// TIA Portal project "Project20" (V19)

(* hardware
DEVICE "S7-1200 station_1"  S7-1200 Station
   slot 0: "Rack_0"  S7-1200 Rack  Rack  V1.0
   slot 1: "PLC_1"  CPU 1215C DC/DC/DC  6ES7 215-1AG40-0XB0  V4.5
*)

// ===== PLC "PLC_1"  CPU 1215C DC/DC/DC =====

VAR_GLOBAL   // PLC tag table "Default tag table"
   "Contactor_Bomba1" AT %Q0.0 : Bool;
   "Contactor_Bomba2" AT %Q0.1 : Bool;
   "Contactor_Bomba3" AT %Q0.2 : Bool;
   "Contactor_Bomba4" AT %Q0.3 : Bool;
   "Contactor_Inyectora" AT %Q0.4 : Bool;
   "Contactor_Bandeja" AT %Q0.5 : Bool;
   "System_Byte" AT %MB1 : Byte;
   "FirstScan" AT %M1.0 : Bool;
   "DiagStatusUpdate" AT %M1.1 : Bool;
   "AlwaysTRUE" AT %M1.2 : Bool;
   "AlwaysFALSE" AT %M1.3 : Bool;
   "Clock_Byte" AT %MB8000 : Byte;
   "Clock_10Hz" AT %M8000.0 : Bool;
   "Clock_5Hz" AT %M8000.1 : Bool;
   "Clock_2.5Hz" AT %M8000.2 : Bool;
   "Clock_2Hz" AT %M8000.3 : Bool;
   "Clock_1.25Hz" AT %M8000.4 : Bool;
   "Clock_1Hz" AT %M8000.5 : Bool;
   "Clock_0.625Hz" AT %M8000.6 : Bool;
   "Clock_0.5Hz" AT %M8000.7 : Bool;
   "Valvula_Entrada_TanqueEntrada" AT %M0.0 : Bool;
   "Valvula_Entrada_TanqueSec1" AT %M0.1 : Bool;
   "Valvula_Entrada_TanqueSec2" AT %M0.2 : Bool;
   "Valvula_Salida_TanqueEntrada" AT %M0.3 : Bool;
   "Valvula_Salida_TanqueSec1" AT %M0.4 : Bool;
   "Valvula_Salida_TanqueSec2" AT %M0.5 : Bool;
   "Pulsador_Bomba1" AT %M0.6 : Bool;
   "Pulsador_Bomba2" AT %M0.7 : Bool;
   "Pulsador_Bomba3" AT %M2.0 : Bool;
   "Pulsador_Bomba4" AT %M2.1 : Bool;
   "Marca_Interruptor" AT %M2.2 : Bool;
   "Marca_Seccionador" AT %M2.3 : Bool;
   "Apertura_Interruptor" AT %M2.4 : Bool;
   "Apertura_Seccionador" AT %M2.5 : Bool;
   "Comando_Llenadora" AT %M2.6 : Bool;
   "Comando_Empacadora" AT %M2.7 : Bool;
END_VAR

TYPE "Datos_Jugos"
VERSION : 0.1
   STRUCT
      Agua : Real;
      Jarabe : Real;
      Manzana : Real;
      Banana : Real;
      Pera : Real;
   END_STRUCT;
END_TYPE

TYPE "Motor_Bomba"
VERSION : 0.1
   STRUCT
      Tension : Array[0..3] of Real;
      Corriente : Real;
      Velocidad : Real;
   END_STRUCT;
END_TYPE

DATA_BLOCK "DB_Llenadora3Botellas"   // DB1
{ S7_Optimized_Access := 'TRUE' }
VERSION : 0.1
// stored: InstanceOfName FB_Llenadora3Botellas
"FB_Llenadora3Botellas"
BEGIN
END_DATA_BLOCK

DATA_BLOCK "DB_Insumos"   // DB8
{ S7_Optimized_Access := 'TRUE' }
VERSION : 0.1
   VAR
      ContajeDinInsumos : Int;
      NivelBotella1 : Int := 0;
      NivelBotella2 : Int := 0;
      NivelBotella3 : Int := 0;
      RecetaActual : Int;
      Jugos : "Datos_Jugos";
   END_VAR
BEGIN
END_DATA_BLOCK

DATA_BLOCK "DB_Fallas"   // DB9
{ S7_Optimized_Access := 'TRUE' }
VERSION : 0.1
BEGIN
END_DATA_BLOCK

DATA_BLOCK "DB_MotorBomba1"   // DB10
{ S7_Optimized_Access := 'TRUE' }
VERSION : 0.1
// stored: InstanceOfName FB_MotorBomba
"FB_MotorBomba"
BEGIN
END_DATA_BLOCK

DATA_BLOCK "DB_MotorBomba2"   // DB11
{ S7_Optimized_Access := 'TRUE' }
VERSION : 0.1
// stored: InstanceOfName FB_MotorBomba
"FB_MotorBomba"
BEGIN
END_DATA_BLOCK

DATA_BLOCK "DB_TanqueEntrada"   // DB12
{ S7_Optimized_Access := 'TRUE' }
VERSION : 0.1
// stored: InstanceOfName FB_Tanque
"FB_Tanque"
BEGIN
END_DATA_BLOCK

DATA_BLOCK "DB_TanqueSec1"   // DB13
{ S7_Optimized_Access := 'TRUE' }
VERSION : 0.1
// stored: InstanceOfName FB_Tanque
"FB_Tanque"
BEGIN
END_DATA_BLOCK

DATA_BLOCK "DB_TanqueSec2"   // DB14
{ S7_Optimized_Access := 'TRUE' }
VERSION : 0.1
// stored: InstanceOfName FB_Tanque
"FB_Tanque"
BEGIN
END_DATA_BLOCK

DATA_BLOCK "DB_MotorBomba3"   // DB15
{ S7_Optimized_Access := 'TRUE' }
VERSION : 0.1
// stored: InstanceOfName FB_MotorBomba
"FB_MotorBomba"
BEGIN
END_DATA_BLOCK

DATA_BLOCK "DB_MotorBomba4"   // DB18
{ S7_Optimized_Access := 'TRUE' }
VERSION : 0.1
// stored: InstanceOfName FB_MotorBomba
"FB_MotorBomba"
BEGIN
END_DATA_BLOCK

DATA_BLOCK "DB_LecturaTensiones"   // DB20
{ S7_Optimized_Access := 'FALSE' }
VERSION : 0.1
   VAR
      Off : Bool;
      Modo : USInt;
      Data_Addr : UDInt := 43020;
      Data_Length : UDInt := 10;
      Connect : TCON_IP_v4;
      Buffer : Array[0..9] of Real;
      TensionSalida : Array[0..2] of Real;
      TensionEscalada : Array[0..5] of Real;
      Accionar_Interruptor : Bool;
      Accionar_Seccionador : Bool;
      Cierre_Interruptor : Bool;
      Cierre_Seccionador : Bool;
      Estado_Interruptor : Bool;
      Estado_Seccionador : Bool;
      ArrayVacio : Array[0..9] of Real;
   END_VAR
BEGIN
   Connect.RemoteAddress.ADDR[1] := 192;
   Connect.RemoteAddress.ADDR[2] := 168;
   Connect.RemoteAddress.ADDR[3] := 13;
   Connect.RemoteAddress.ADDR[4] := 68;
   Connect.InterfaceId := 64;
   Connect.ID := 1;
   Connect.ConnectionType := 11;
   Connect.ActiveEstablished := TRUE;
   Connect.RemotePort := 502;
END_DATA_BLOCK

DATA_BLOCK "DB_LecturaMotores"   // DB21
{ S7_Optimized_Access := 'TRUE' }
VERSION : 0.1
   VAR
      MotorBomba1 : "Motor_Bomba";
      MotorBomba2 : "Motor_Bomba";
      MotorBomba3 : "Motor_Bomba";
      MotorBomba4 : "Motor_Bomba";
      Angulo : Int;
      TensionSalida : Array[0..2] of Real;
   END_VAR
BEGIN
END_DATA_BLOCK

DATA_BLOCK "DB_LecturaMedidor"   // DB38
{ S7_Optimized_Access := 'FALSE' }
VERSION : 0.1
// stored: InstanceOfName FB_LecturaMedidor
"FB_LecturaMedidor"
BEGIN
END_DATA_BLOCK

DATA_BLOCK "DB_LecturaCorrientes"   // DB39
{ S7_Optimized_Access := 'FALSE' }
VERSION : 0.1
   VAR
      Off : Bool;
      Modo : USInt;
      Data_Addr : UDInt := 43000;
      Data_Length : UDInt := 10;
      Connect : TCON_IP_v4;
      Buffer : Array[0..9] of Real;
   END_VAR
BEGIN
   Connect.RemoteAddress.ADDR[1] := 192;
   Connect.RemoteAddress.ADDR[2] := 168;
   Connect.RemoteAddress.ADDR[3] := 13;
   Connect.RemoteAddress.ADDR[4] := 68;
   Connect.InterfaceId := 64;
   Connect.ID := 2;
   Connect.ConnectionType := 11;
   Connect.ActiveEstablished := TRUE;
   Connect.RemotePort := 502;
END_DATA_BLOCK

DATA_BLOCK "DB_SimEmpacado"   // DB40
{ S7_Optimized_Access := 'TRUE' }
VERSION : 0.1
// stored: InstanceOfName FB_SimEmpacado
"FB_SimEmpacado"
BEGIN
END_DATA_BLOCK

// folder: System blocks/Program resources

DATA_BLOCK "Contador_Botella1"   // DB2
{ S7_Optimized_Access := 'TRUE' }
AUTHOR : Simatic
FAMILY : IEC
NAME : CNTR
VERSION : 1.0
// stored: InstanceOfName IEC_COUNTER
"IEC_COUNTER"
BEGIN
END_DATA_BLOCK

DATA_BLOCK "TON_DelayCajas"   // DB3
{ S7_Optimized_Access := 'TRUE' }
AUTHOR : Simatic
FAMILY : IEC
NAME : IEC_TMR
VERSION : 1.0
// stored: InstanceOfName IEC_TIMER
"IEC_TIMER"
BEGIN
END_DATA_BLOCK

DATA_BLOCK "Contador_Botella2"   // DB4
{ S7_Optimized_Access := 'TRUE' }
AUTHOR : Simatic
FAMILY : IEC
NAME : CNTR
VERSION : 1.0
// stored: InstanceOfName IEC_COUNTER
"IEC_COUNTER"
BEGIN
END_DATA_BLOCK

DATA_BLOCK "Contador_Botella3"   // DB5
{ S7_Optimized_Access := 'TRUE' }
AUTHOR : Simatic
FAMILY : IEC
NAME : CNTR
VERSION : 1.0
// stored: InstanceOfName IEC_COUNTER
"IEC_COUNTER"
BEGIN
END_DATA_BLOCK

DATA_BLOCK "Timer_Bandeja_Llenadora"   // DB6
{ S7_Optimized_Access := 'TRUE' }
AUTHOR : Simatic
FAMILY : IEC
NAME : IEC_TMR
VERSION : 1.0
// stored: InstanceOfName IEC_TIMER
"IEC_TIMER"
BEGIN
END_DATA_BLOCK

DATA_BLOCK "Timer_Vaciado_Tanque"   // DB7
{ S7_Optimized_Access := 'TRUE' }
AUTHOR : Simatic
FAMILY : IEC
NAME : IEC_TMR
VERSION : 1.0
// stored: InstanceOfName IEC_TIMER
"IEC_TIMER"
BEGIN
END_DATA_BLOCK

DATA_BLOCK "Timer_Llenado_Tanque"   // DB16
{ S7_Optimized_Access := 'TRUE' }
AUTHOR : Simatic
FAMILY : IEC
NAME : IEC_TMR
VERSION : 1.0
// stored: InstanceOfName IEC_TIMER
"IEC_TIMER"
BEGIN
END_DATA_BLOCK

DATA_BLOCK "Contador_Tanque"   // DB17
{ S7_Optimized_Access := 'TRUE' }
AUTHOR : Simatic
FAMILY : IEC
NAME : CNTR
VERSION : 1.0
// stored: InstanceOfName IEC_COUNTER
"IEC_COUNTER"
BEGIN
END_DATA_BLOCK

DATA_BLOCK "Timer_Apagado_Bandeja"   // DB22
{ S7_Optimized_Access := 'TRUE' }
AUTHOR : Simatic
FAMILY : IEC
NAME : IEC_TMR
VERSION : 1.0
// stored: InstanceOfName IEC_TIMER
"IEC_TIMER"
BEGIN
END_DATA_BLOCK

DATA_BLOCK "Timer_Delay_Realista"   // DB23
{ S7_Optimized_Access := 'TRUE' }
AUTHOR : Simatic
FAMILY : IEC
NAME : IEC_TMR
VERSION : 1.0
// stored: InstanceOfName IEC_TIMER
"IEC_TIMER"
BEGIN
END_DATA_BLOCK

DATA_BLOCK "Timer_Delay_Realista_2"   // DB24
{ S7_Optimized_Access := 'TRUE' }
AUTHOR : Simatic
FAMILY : IEC
NAME : IEC_TMR
VERSION : 1.0
// stored: InstanceOfName IEC_TIMER
"IEC_TIMER"
BEGIN
END_DATA_BLOCK

DATA_BLOCK "Timer_Din_Tanques_3s"   // DB28
{ S7_Optimized_Access := 'TRUE' }
AUTHOR : Simatic
FAMILY : IEC
NAME : IEC_TMR
VERSION : 1.0
// stored: InstanceOfName IEC_TIMER
"IEC_TIMER"
BEGIN
END_DATA_BLOCK

DATA_BLOCK "Timer_Din_Tanques_7s"   // DB29
{ S7_Optimized_Access := 'TRUE' }
AUTHOR : Simatic
FAMILY : IEC
NAME : IEC_TMR
VERSION : 1.0
// stored: InstanceOfName IEC_TIMER
"IEC_TIMER"
BEGIN
END_DATA_BLOCK

DATA_BLOCK "Timer_Din_Tanques_10s"   // DB30
{ S7_Optimized_Access := 'TRUE' }
AUTHOR : Simatic
FAMILY : IEC
NAME : IEC_TMR
VERSION : 1.0
// stored: InstanceOfName IEC_TIMER
"IEC_TIMER"
BEGIN
END_DATA_BLOCK

DATA_BLOCK "Timer_Din_Tanques_20s"   // DB31
{ S7_Optimized_Access := 'TRUE' }
AUTHOR : Simatic
FAMILY : IEC
NAME : IEC_TMR
VERSION : 1.0
// stored: InstanceOfName IEC_TIMER
"IEC_TIMER"
BEGIN
END_DATA_BLOCK

DATA_BLOCK "Timer_Din_Tanques_30s"   // DB32
{ S7_Optimized_Access := 'TRUE' }
AUTHOR : Simatic
FAMILY : IEC
NAME : IEC_TMR
VERSION : 1.0
// stored: InstanceOfName IEC_TIMER
"IEC_TIMER"
BEGIN
END_DATA_BLOCK

DATA_BLOCK "Timer_Din_Tanques_40s"   // DB33
{ S7_Optimized_Access := 'TRUE' }
AUTHOR : Simatic
FAMILY : IEC
NAME : IEC_TMR
VERSION : 1.0
// stored: InstanceOfName IEC_TIMER
"IEC_TIMER"
BEGIN
END_DATA_BLOCK

DATA_BLOCK "Timer_Din_Tanques_15s"   // DB34
{ S7_Optimized_Access := 'TRUE' }
AUTHOR : Simatic
FAMILY : IEC
NAME : IEC_TMR
VERSION : 1.0
// stored: InstanceOfName IEC_TIMER
"IEC_TIMER"
BEGIN
END_DATA_BLOCK

DATA_BLOCK "Timer_Din_Tanques_25s"   // DB35
{ S7_Optimized_Access := 'TRUE' }
AUTHOR : Simatic
FAMILY : IEC
NAME : IEC_TMR
VERSION : 1.0
// stored: InstanceOfName IEC_TIMER
"IEC_TIMER"
BEGIN
END_DATA_BLOCK

DATA_BLOCK "Timer_Din_Tanques_35s"   // DB36
{ S7_Optimized_Access := 'TRUE' }
AUTHOR : Simatic
FAMILY : IEC
NAME : IEC_TMR
VERSION : 1.0
// stored: InstanceOfName IEC_TIMER
"IEC_TIMER"
BEGIN
END_DATA_BLOCK

// folder: (top level)

FUNCTION_BLOCK "FB_MotorBomba"   // FB1, LAD
{ S7_Optimized_Access := 'TRUE' }
VERSION : 0.1
   VAR_INPUT
      Comando : Bool;
      TensionL1 : Real;
      TensionL2 : Real;
      TensionL3 : Real;
      EntVel : Real;
      EntCorr : Real;
      Reset : Bool;
      Factor : Real := 2.2;
   END_VAR
   VAR_OUTPUT
      Contactor : Bool;
      TensionR1 : Real;
      TensionR2 : Real;
      TensionR3 : Real;
      TensionProm : Real;
      VelSal : Real;
      CorrSal : Real;
      Trip : Bool;
      Estado : Int := 0;
   END_VAR
   VAR
      EstadoComando : Bool := false;
      EstadoBomba : Int := 0;
   END_VAR
   VAR CONSTANT
      DIV : Int := 3;
   END_VAR
   VAR_TEMP   // added for the SCL form of the ladder/FBD networks
      _w1 : Bool;
   END_VAR
BEGIN

REGION Network 1
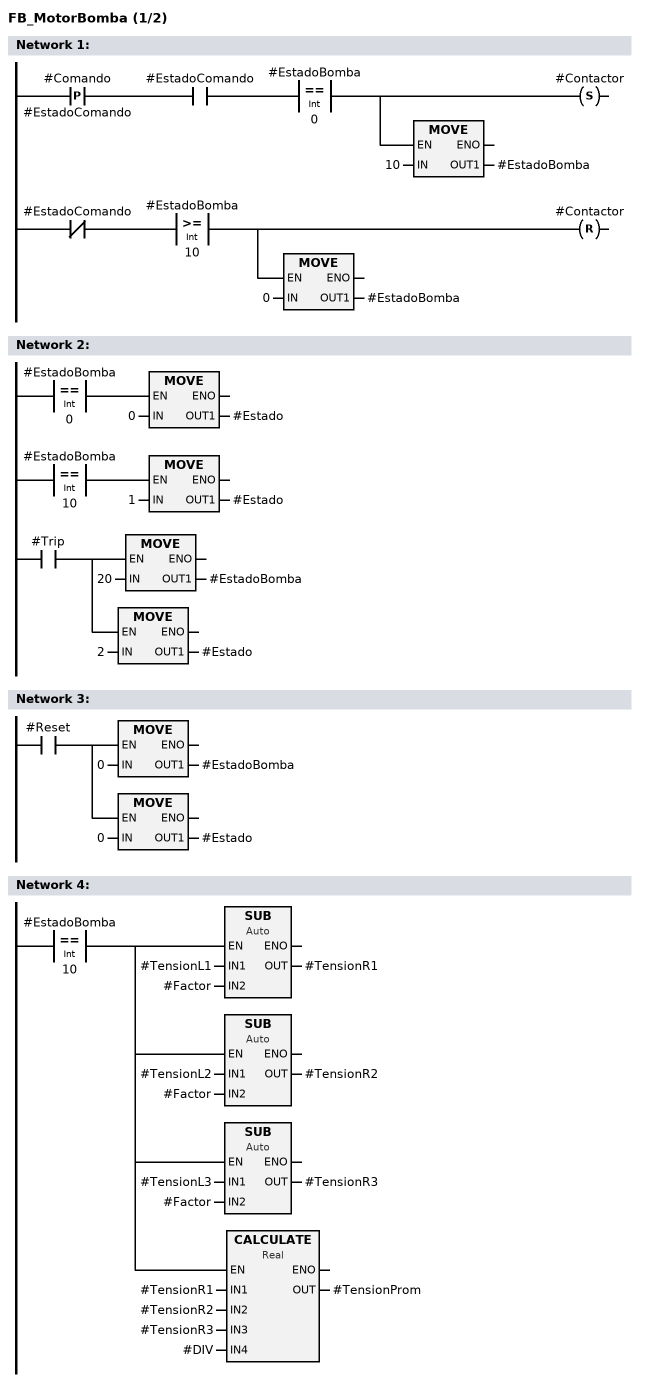
   RUNG wire#powerrail
      P_Contact(operand := #Comando, bit := #EstadoComando)
      Contact( #EstadoComando )
      { S7_Templates := "SrcType := Int" } EQ_Contact(in1 := #EstadoBomba, in2 := 0)
      wire#w1
      S_Coil( #Contactor )
   END_RUNG
   RUNG wire#w1
      Move(in := 10, out1 => #EstadoBomba)
   END_RUNG
   RUNG wire#powerrail
      I_Contact( #EstadoComando )
      { S7_Templates := "SrcType := Int" } GE_Contact(in1 := #EstadoBomba, in2 := 10)
      wire#w2
      R_Coil( #Contactor )
   END_RUNG
   RUNG wire#w2
      Move(in := 0, out1 => #EstadoBomba)
   END_RUNG
   // the same network as SCL:
   #_w1 := #Comando AND NOT #EstadoComando;   // rising edge of #Comando
   #EstadoComando := #Comando;
   IF #_w1 AND #EstadoComando AND (#EstadoBomba = 0) THEN
       #Contactor := TRUE;
       #EstadoBomba := 10;
   END_IF;
   IF NOT #EstadoComando AND (#EstadoBomba >= 10) THEN
       #Contactor := FALSE;
       #EstadoBomba := 0;
   END_IF;
END_REGION

REGION Network 2
   RUNG wire#powerrail
      { S7_Templates := "SrcType := Int" } EQ_Contact(in1 := #EstadoBomba, in2 := 0)
      Move(in := 0, out1 => #Estado)
   END_RUNG
   RUNG wire#powerrail
      { S7_Templates := "SrcType := Int" } EQ_Contact(in1 := #EstadoBomba, in2 := 10)
      Move(in := 1, out1 => #Estado)
   END_RUNG
   RUNG wire#powerrail
      Contact( #Trip )
      wire#w1
      Move(in := 20, out1 => #EstadoBomba)
   END_RUNG
   RUNG wire#w1
      Move(in := 2, out1 => #Estado)
   END_RUNG
   // the same network as SCL:
   IF #EstadoBomba = 0 THEN #Estado := 0; END_IF;
   IF #EstadoBomba = 10 THEN #Estado := 1; END_IF;
   IF #Trip THEN
       #EstadoBomba := 20;
       #Estado := 2;
   END_IF;
END_REGION

REGION Network 3
   RUNG wire#powerrail
      Contact( #Reset )
      wire#w1
      Move(in := 0, out1 => #EstadoBomba)
   END_RUNG
   RUNG wire#w1
      Move(in := 0, out1 => #Estado)
   END_RUNG
   // the same network as SCL:
   IF #Reset THEN
       #EstadoBomba := 0;
       #Estado := 0;
   END_IF;
END_REGION

REGION Network 4
   RUNG wire#powerrail
      { S7_Templates := "SrcType := Int" } EQ_Contact(in1 := #EstadoBomba, in2 := 10)
      wire#w1
      Sub(in1 := #TensionL1, in2 := #Factor, out => #TensionR1)
   END_RUNG
   RUNG wire#w1
      Sub(in1 := #TensionL2, in2 := #Factor, out => #TensionR2)
   END_RUNG
   RUNG wire#w1
      Sub(in1 := #TensionL3, in2 := #Factor, out => #TensionR3)
   END_RUNG
   RUNG wire#w1
      { S7_Templates := "SrcType := Real"; S7_Expression := "(IN1+IN2+IN3)/(IN4)" } Calculate(in1 := #TensionR1, in2 := #TensionR2, in3 := #TensionR3, in4 := #DIV, out => #TensionProm)
   END_RUNG
   // the same network as SCL:
   IF #EstadoBomba = 10 THEN
       #TensionR1 := #TensionL1 - #Factor;
       #TensionR2 := #TensionL2 - #Factor;
       #TensionR3 := #TensionL3 - #Factor;
       #TensionProm := (#TensionR1+#TensionR2+#TensionR3)/(#DIV);
   END_IF;
END_REGION

REGION Network 5
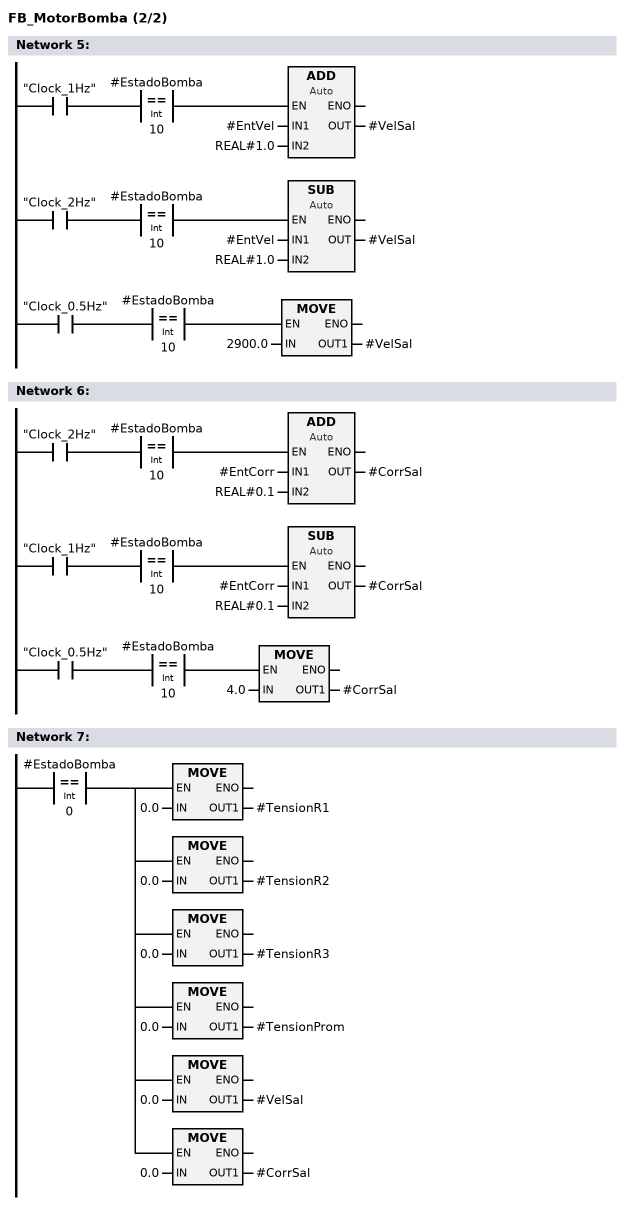
   RUNG wire#powerrail
      Contact( "Clock_1Hz" )
      { S7_Templates := "SrcType := Int" } EQ_Contact(in1 := #EstadoBomba, in2 := 10)
      Add(in1 := #EntVel, in2 := REAL#1.0, out => #VelSal)
   END_RUNG
   RUNG wire#powerrail
      Contact( "Clock_2Hz" )
      { S7_Templates := "SrcType := Int" } EQ_Contact(in1 := #EstadoBomba, in2 := 10)
      Sub(in1 := #EntVel, in2 := REAL#1.0, out => #VelSal)
   END_RUNG
   RUNG wire#powerrail
      Contact( "Clock_0.5Hz" )
      { S7_Templates := "SrcType := Int" } EQ_Contact(in1 := #EstadoBomba, in2 := 10)
      Move(in := 2900.0, out1 => #VelSal)
   END_RUNG
   // the same network as SCL:
   IF "Clock_1Hz" AND (#EstadoBomba = 10) THEN #VelSal := #EntVel + REAL#1.0; END_IF;
   IF "Clock_2Hz" AND (#EstadoBomba = 10) THEN #VelSal := #EntVel - REAL#1.0; END_IF;
   IF "Clock_0.5Hz" AND (#EstadoBomba = 10) THEN #VelSal := 2900.0; END_IF;
END_REGION

REGION Network 6
   RUNG wire#powerrail
      Contact( "Clock_2Hz" )
      { S7_Templates := "SrcType := Int" } EQ_Contact(in1 := #EstadoBomba, in2 := 10)
      Add(in1 := #EntCorr, in2 := REAL#0.1, out => #CorrSal)
   END_RUNG
   RUNG wire#powerrail
      Contact( "Clock_1Hz" )
      { S7_Templates := "SrcType := Int" } EQ_Contact(in1 := #EstadoBomba, in2 := 10)
      Sub(in1 := #EntCorr, in2 := REAL#0.1, out => #CorrSal)
   END_RUNG
   RUNG wire#powerrail
      Contact( "Clock_0.5Hz" )
      { S7_Templates := "SrcType := Int" } EQ_Contact(in1 := #EstadoBomba, in2 := 10)
      Move(in := 4.0, out1 => #CorrSal)
   END_RUNG
   // the same network as SCL:
   IF "Clock_2Hz" AND (#EstadoBomba = 10) THEN #CorrSal := #EntCorr + REAL#0.1; END_IF;
   IF "Clock_1Hz" AND (#EstadoBomba = 10) THEN #CorrSal := #EntCorr - REAL#0.1; END_IF;
   IF "Clock_0.5Hz" AND (#EstadoBomba = 10) THEN #CorrSal := 4.0; END_IF;
END_REGION

REGION Network 7
   RUNG wire#powerrail
      { S7_Templates := "SrcType := Int" } EQ_Contact(in1 := #EstadoBomba, in2 := 0)
      wire#w1
      Move(in := 0.0, out1 => #TensionR1)
   END_RUNG
   RUNG wire#w1
      Move(in := 0.0, out1 => #TensionR2)
   END_RUNG
   RUNG wire#w1
      Move(in := 0.0, out1 => #TensionR3)
   END_RUNG
   RUNG wire#w1
      Move(in := 0.0, out1 => #TensionProm)
   END_RUNG
   RUNG wire#w1
      Move(in := 0.0, out1 => #VelSal)
   END_RUNG
   RUNG wire#w1
      Move(in := 0.0, out1 => #CorrSal)
   END_RUNG
   // the same network as SCL:
   IF #EstadoBomba = 0 THEN
       #TensionR1 := 0.0;
       #TensionR2 := 0.0;
       #TensionR3 := 0.0;
       #TensionProm := 0.0;
       #VelSal := 0.0;
       #CorrSal := 0.0;
   END_IF;
END_REGION
END_FUNCTION_BLOCK

FUNCTION_BLOCK "FB_Llenadora3Botellas"   // FB2, LAD
{ S7_Optimized_Access := 'TRUE' }
VERSION : 0.1
   VAR_INPUT
      Comando : Bool;
      Setpoint : Real := 0.0;
      SetActual : Int;
   END_VAR
   VAR_OUTPUT
      ContactorBandeja : Bool;
      ContactorInyectora : Bool;
      Estado : Int;
      NivelBotella1 : Int;
      NivelBotella2 : Int;
      NivelBotella3 : Int;
   END_VAR
   VAR
      EstadoComando : Bool;
      DesplazarBotellas : Bool;
      EstadoLlenadora : Int := 0;
      SetpointInt : Int;
      ResetContadores : Bool;
   END_VAR
   VAR RETAIN
      Contador_BotellasManzana : CTU_INT;
      Contador_BotellasBanana : CTU_INT;
      Contador_BotellasPera : CTU_INT;
      Contador_BotellasMulti : CTU_INT;
      ActivarResetBotellas : Int := 10000;
      ResetBotellas : Bool;
   END_VAR
   VAR_TEMP   // added for the SCL form of the ladder/FBD networks
      _w1 : Bool;
   END_VAR
BEGIN

REGION Network 1
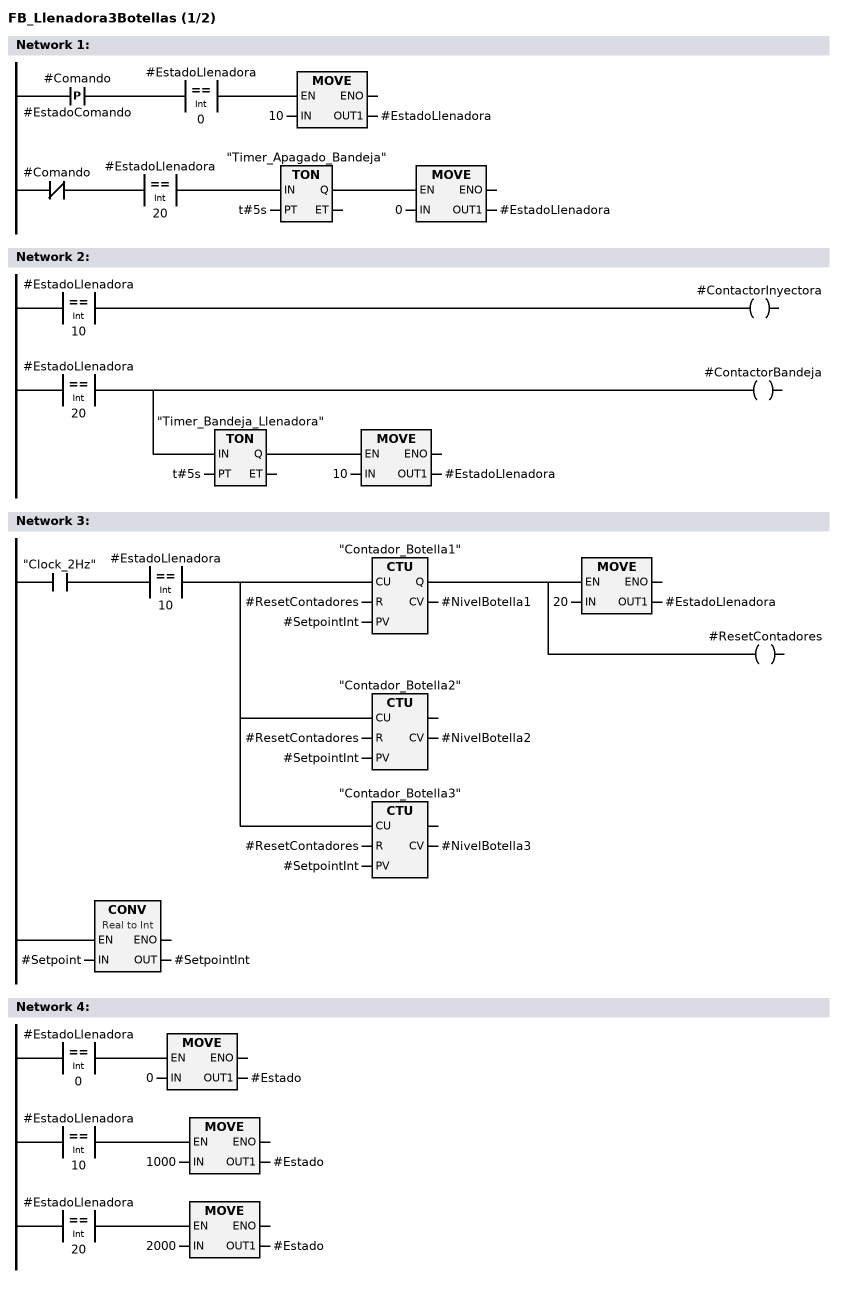
   #_w1 := #Comando AND NOT #EstadoComando;   // rising edge of #Comando
   #EstadoComando := #Comando;
   IF #_w1 AND (#EstadoLlenadora = 0) THEN #EstadoLlenadora := 10; END_IF;
   "Timer_Apagado_Bandeja".TON(IN := NOT #Comando AND (#EstadoLlenadora = 20), PT := t#5s);
   IF "Timer_Apagado_Bandeja".Q THEN #EstadoLlenadora := 0; END_IF;
END_REGION

REGION Network 2
   #ContactorInyectora := #EstadoLlenadora = 10;
   #ContactorBandeja := #EstadoLlenadora = 20;
   "Timer_Bandeja_Llenadora".TON(IN := #ContactorBandeja, PT := t#5s);
   IF "Timer_Bandeja_Llenadora".Q THEN #EstadoLlenadora := 10; END_IF;
END_REGION

REGION Network 3
   #_w1 := "Clock_2Hz" AND (#EstadoLlenadora = 10);
   "Contador_Botella1".CTU(CU := #_w1, R := #ResetContadores, PV := #SetpointInt, CV => #NivelBotella1);
   IF "Contador_Botella1".Q THEN #EstadoLlenadora := 20; END_IF;
   #ResetContadores := "Contador_Botella1".Q;
   "Contador_Botella2".CTU(CU := #_w1, R := #ResetContadores, PV := #SetpointInt, CV => #NivelBotella2);
   "Contador_Botella3".CTU(CU := #_w1, R := #ResetContadores, PV := #SetpointInt, CV => #NivelBotella3);
   #SetpointInt := REAL_TO_INT(#Setpoint);
END_REGION

REGION Network 4
   RUNG wire#powerrail
      { S7_Templates := "SrcType := Int" } EQ_Contact(in1 := #EstadoLlenadora, in2 := 0)
      Move(in := 0, out1 => #Estado)
   END_RUNG
   RUNG wire#powerrail
      { S7_Templates := "SrcType := Int" } EQ_Contact(in1 := #EstadoLlenadora, in2 := 10)
      Move(in := 1000, out1 => #Estado)
   END_RUNG
   RUNG wire#powerrail
      { S7_Templates := "SrcType := Int" } EQ_Contact(in1 := #EstadoLlenadora, in2 := 20)
      Move(in := 2000, out1 => #Estado)
   END_RUNG
   // the same network as SCL:
   IF #EstadoLlenadora = 0 THEN #Estado := 0; END_IF;
   IF #EstadoLlenadora = 10 THEN #Estado := 1000; END_IF;
   IF #EstadoLlenadora = 20 THEN #Estado := 2000; END_IF;
END_REGION

REGION Network 5
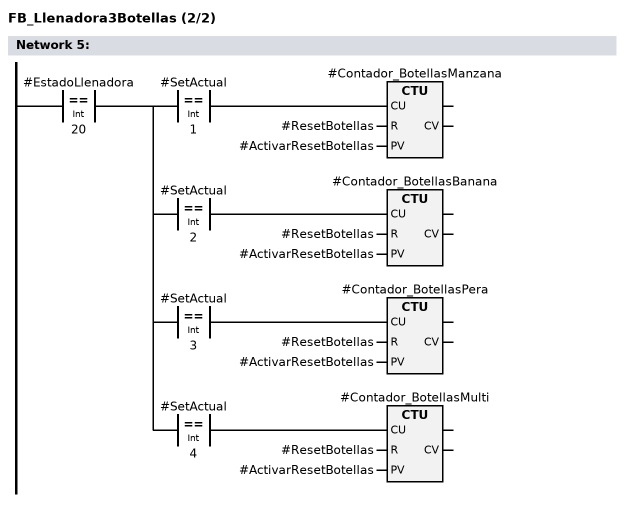
   #_w1 := #EstadoLlenadora = 20;
   #Contador_BotellasManzana(CU := #_w1 AND (#SetActual = 1), R := #ResetBotellas, PV := #ActivarResetBotellas);   // CTU
   #Contador_BotellasBanana(CU := #_w1 AND (#SetActual = 2), R := #ResetBotellas, PV := #ActivarResetBotellas);   // CTU
   #Contador_BotellasPera(CU := #_w1 AND (#SetActual = 3), R := #ResetBotellas, PV := #ActivarResetBotellas);   // CTU
   #Contador_BotellasMulti(CU := #_w1 AND (#SetActual = 4), R := #ResetBotellas, PV := #ActivarResetBotellas);   // CTU
END_REGION
END_FUNCTION_BLOCK

FUNCTION_BLOCK "FB_Tanque"   // FB4, LAD
{ S7_Optimized_Access := 'TRUE' }
VERSION : 0.1
   VAR_INPUT
      ValvulaEntrada : Bool;
      SetpointLlenado : Int := 90;
      ValvulaSalida : Bool;
      SetpointVaciado : Int := 10;
      PresionEntrada : Real;
      TemperaturaEntrada : Real;
      HumedadEntrada : Real;
      TipoTanque : Int;
   END_VAR
   VAR_OUTPUT
      Nivel : Int;
      PresionSalida : Real;
      TemperaturaSalida : Real;
      HumedadSalida : Real;
      AlarmaRebase : Bool;
   END_VAR
   VAR
      TimerVaciado : Bool;
      TimerLlenado : Bool;
      Estado : Int := 0;
      TiempoLlenado : Time;
      TiempoVaciado : Time;
      Reset13sP : Bool;
      Reset17sP : Bool;
      Reset22sP : Bool;
      Reset20sT : Bool;
      Reset30sT : Bool;
      Reset40sT : Bool;
      Reset15sH : Bool;
      Reset25sH : Bool;
      Reset35sH : Bool;
   END_VAR
BEGIN

REGION Network 1
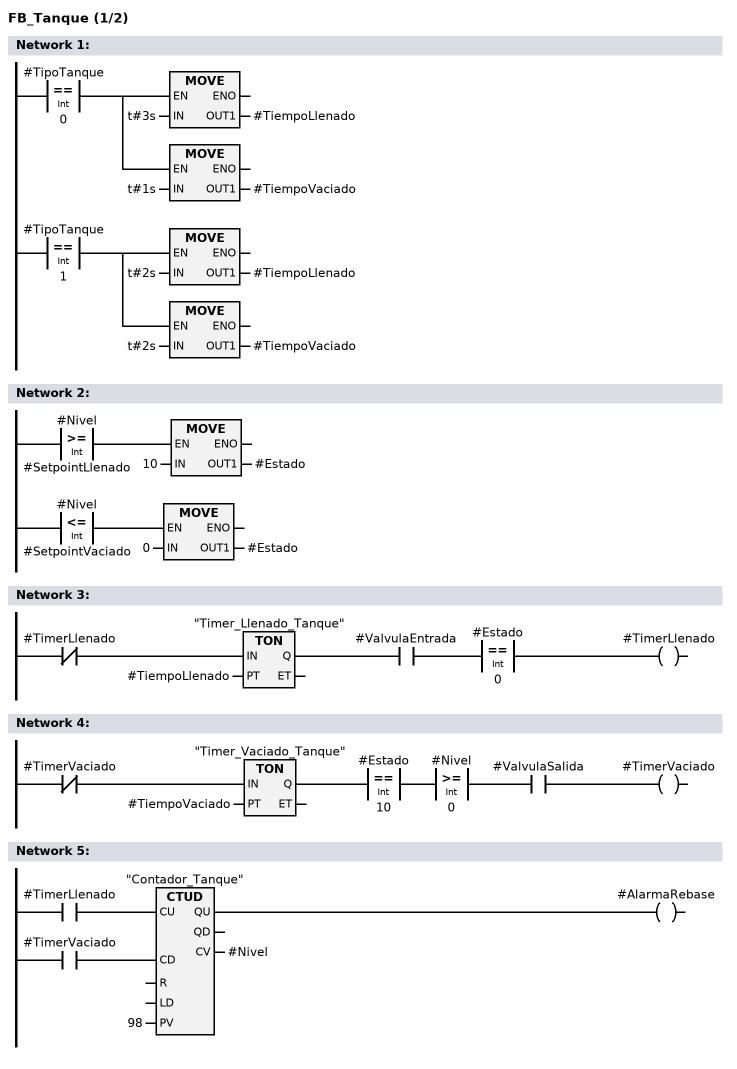
   RUNG wire#powerrail
      { S7_Templates := "SrcType := Int" } EQ_Contact(in1 := #TipoTanque, in2 := 0)
      wire#w1
      Move(in := t#3s, out1 => #TiempoLlenado)
   END_RUNG
   RUNG wire#w1
      Move(in := t#1s, out1 => #TiempoVaciado)
   END_RUNG
   RUNG wire#powerrail
      { S7_Templates := "SrcType := Int" } EQ_Contact(in1 := #TipoTanque, in2 := 1)
      wire#w2
      Move(in := t#2s, out1 => #TiempoLlenado)
   END_RUNG
   RUNG wire#w2
      Move(in := t#2s, out1 => #TiempoVaciado)
   END_RUNG
   // the same network as SCL:
   IF #TipoTanque = 0 THEN
       #TiempoLlenado := t#3s;
       #TiempoVaciado := t#1s;
   END_IF;
   IF #TipoTanque = 1 THEN
       #TiempoLlenado := t#2s;
       #TiempoVaciado := t#2s;
   END_IF;
END_REGION

REGION Network 2
   RUNG wire#powerrail
      { S7_Templates := "SrcType := Int" } GE_Contact(in1 := #Nivel, in2 := #SetpointLlenado)
      Move(in := 10, out1 => #Estado)
   END_RUNG
   RUNG wire#powerrail
      { S7_Templates := "SrcType := Int" } LE_Contact(in1 := #Nivel, in2 := #SetpointVaciado)
      Move(in := 0, out1 => #Estado)
   END_RUNG
   // the same network as SCL:
   IF #Nivel >= #SetpointLlenado THEN #Estado := 10; END_IF;
   IF #Nivel <= #SetpointVaciado THEN #Estado := 0; END_IF;
END_REGION

REGION Network 3
   "Timer_Llenado_Tanque".TON(IN := NOT #TimerLlenado, PT := #TiempoLlenado);
   #TimerLlenado := "Timer_Llenado_Tanque".Q AND #ValvulaEntrada AND (#Estado = 0);
END_REGION

REGION Network 4
   "Timer_Vaciado_Tanque".TON(IN := NOT #TimerVaciado, PT := #TiempoVaciado);
   #TimerVaciado := "Timer_Vaciado_Tanque".Q AND (#Estado = 10) AND (#Nivel >= 0) AND #ValvulaSalida;
END_REGION

REGION Network 5
   "Contador_Tanque".CTUD(CU := #TimerLlenado, CD := #TimerVaciado, PV := 98, CV => #Nivel);
   #AlarmaRebase := "Contador_Tanque".QU;
END_REGION

REGION Network 6
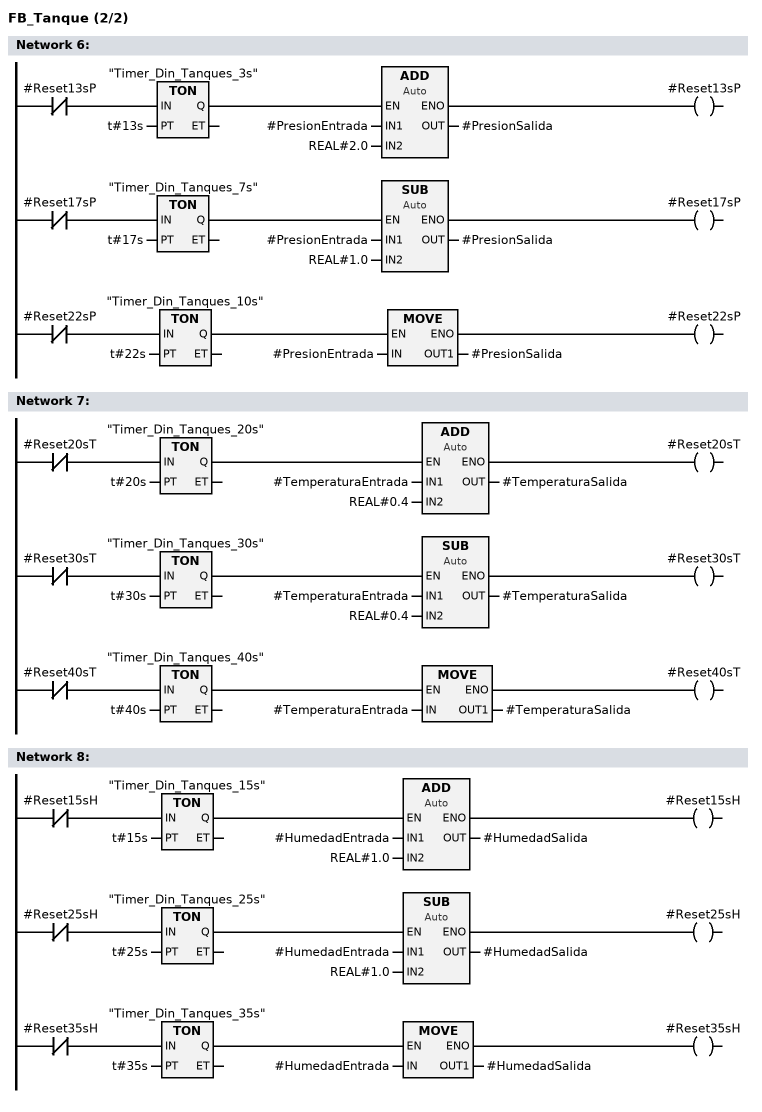
   "Timer_Din_Tanques_3s".TON(IN := NOT #Reset13sP, PT := t#13s);
   IF "Timer_Din_Tanques_3s".Q THEN #PresionSalida := #PresionEntrada + REAL#2.0; END_IF;
   #Reset13sP := "Timer_Din_Tanques_3s".Q;
   "Timer_Din_Tanques_7s".TON(IN := NOT #Reset17sP, PT := t#17s);
   IF "Timer_Din_Tanques_7s".Q THEN #PresionSalida := #PresionEntrada - REAL#1.0; END_IF;
   #Reset17sP := "Timer_Din_Tanques_7s".Q;
   "Timer_Din_Tanques_10s".TON(IN := NOT #Reset22sP, PT := t#22s);
   IF "Timer_Din_Tanques_10s".Q THEN #PresionSalida := #PresionEntrada; END_IF;
   #Reset22sP := "Timer_Din_Tanques_10s".Q;
END_REGION

REGION Network 7
   "Timer_Din_Tanques_20s".TON(IN := NOT #Reset20sT, PT := t#20s);
   IF "Timer_Din_Tanques_20s".Q THEN #TemperaturaSalida := #TemperaturaEntrada + REAL#0.4; END_IF;
   #Reset20sT := "Timer_Din_Tanques_20s".Q;
   "Timer_Din_Tanques_30s".TON(IN := NOT #Reset30sT, PT := t#30s);
   IF "Timer_Din_Tanques_30s".Q THEN #TemperaturaSalida := #TemperaturaEntrada - REAL#0.4; END_IF;
   #Reset30sT := "Timer_Din_Tanques_30s".Q;
   "Timer_Din_Tanques_40s".TON(IN := NOT #Reset40sT, PT := t#40s);
   IF "Timer_Din_Tanques_40s".Q THEN #TemperaturaSalida := #TemperaturaEntrada; END_IF;
   #Reset40sT := "Timer_Din_Tanques_40s".Q;
END_REGION

REGION Network 8
   "Timer_Din_Tanques_15s".TON(IN := NOT #Reset15sH, PT := t#15s);
   IF "Timer_Din_Tanques_15s".Q THEN #HumedadSalida := #HumedadEntrada + REAL#1.0; END_IF;
   #Reset15sH := "Timer_Din_Tanques_15s".Q;
   "Timer_Din_Tanques_25s".TON(IN := NOT #Reset25sH, PT := t#25s);
   IF "Timer_Din_Tanques_25s".Q THEN #HumedadSalida := #HumedadEntrada - REAL#1.0; END_IF;
   #Reset25sH := "Timer_Din_Tanques_25s".Q;
   "Timer_Din_Tanques_35s".TON(IN := NOT #Reset35sH, PT := t#35s);
   IF "Timer_Din_Tanques_35s".Q THEN #HumedadSalida := #HumedadEntrada; END_IF;
   #Reset35sH := "Timer_Din_Tanques_35s".Q;
END_REGION
END_FUNCTION_BLOCK

FUNCTION_BLOCK "FB_LecturaMedidor"   // FB5, LAD
{ S7_Optimized_Access := 'FALSE' }
VERSION : 0.1
   VAR_INPUT
      Encendido : Bool;
   END_VAR
   VAR
      MB_CLIENT_LecturaMedidor : MB_CLIENT;
      ArrayVacio : Array[0..7] of Real;
      Buffer : Array[0..7] of Real;
      OrdenDato : Int;
      Connect : TCON_IP_v4;
      Timer_LecturaMedidor : TON_TIME;
      Data_Addr : UDInt;
      Modo : USInt;
      Data_Len : UDInt := 2;
      Off : Bool;
      ResetTimer : Bool;
   END_VAR
   // Connect.InterfaceId := 64;
   // Connect.ID := 3;
   // Connect.ConnectionType := 11;
   // Connect.ActiveEstablished := TRUE;
   // Connect.RemoteAddress.ADDR[1] := 192;
   // Connect.RemoteAddress.ADDR[2] := 168;
   // Connect.RemoteAddress.ADDR[3] := 13;
   // Connect.RemoteAddress.ADDR[4] := 68;
   // Connect.RemotePort := 502;
BEGIN

REGION Network 1
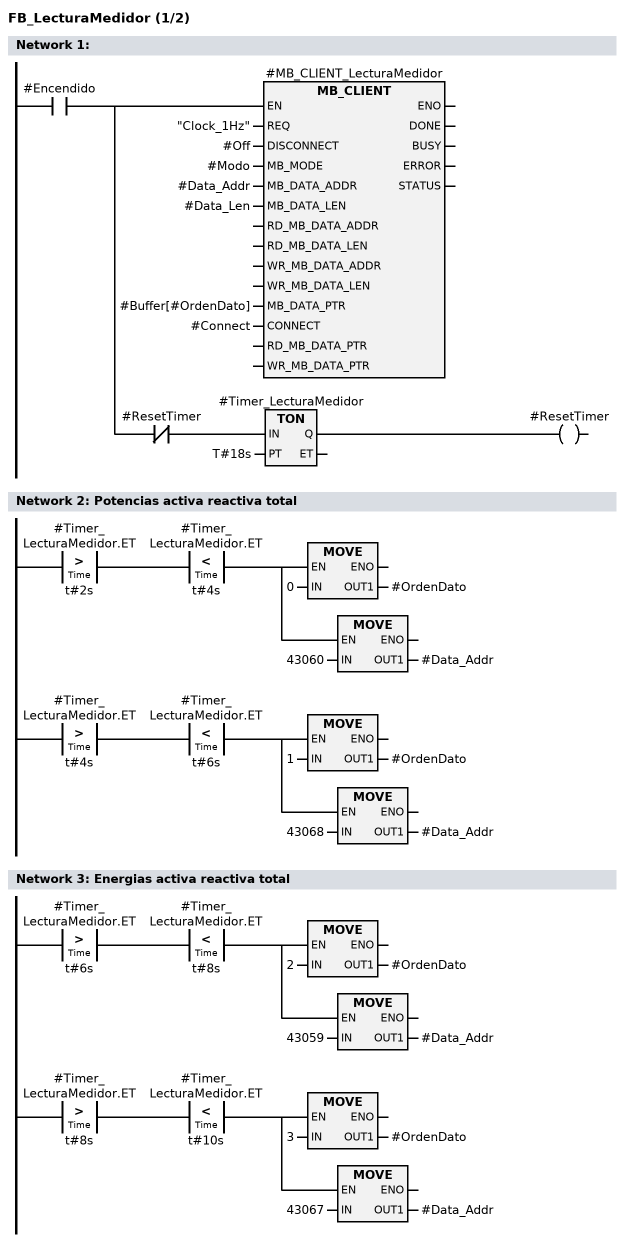
   IF #Encendido THEN
       #MB_CLIENT_LecturaMedidor(REQ := "Clock_1Hz",   // MB_CLIENT
                               DISCONNECT := #Off,
                               MB_MODE := #Modo,
                               MB_DATA_ADDR := #Data_Addr,
                               MB_DATA_LEN := #Data_Len,
                               MB_DATA_PTR := #Buffer[#OrdenDato],
                               CONNECT := #Connect);
   END_IF;
   #Timer_LecturaMedidor(IN := #Encendido AND NOT #ResetTimer, PT := T#18s);   // TON
   #ResetTimer := #Timer_LecturaMedidor.Q;
END_REGION

REGION Network 2: Potencias activa reactiva total
   RUNG wire#powerrail
      { S7_Templates := "SrcType := Time" } GT_Contact(in1 := #Timer_LecturaMedidor.ET, in2 := t#2s)
      { S7_Templates := "SrcType := Time" } LT_Contact(in1 := #Timer_LecturaMedidor.ET, in2 := t#4s)
      wire#w1
      Move(in := 0, out1 => #OrdenDato)
   END_RUNG
   RUNG wire#w1
      Move(in := 43060, out1 => #Data_Addr)
   END_RUNG
   RUNG wire#powerrail
      { S7_Templates := "SrcType := Time" } GT_Contact(in1 := #Timer_LecturaMedidor.ET, in2 := t#4s)
      { S7_Templates := "SrcType := Time" } LT_Contact(in1 := #Timer_LecturaMedidor.ET, in2 := t#6s)
      wire#w2
      Move(in := 1, out1 => #OrdenDato)
   END_RUNG
   RUNG wire#w2
      Move(in := 43068, out1 => #Data_Addr)
   END_RUNG
   // the same network as SCL:
   IF (#Timer_LecturaMedidor.ET > t#2s) AND (#Timer_LecturaMedidor.ET < t#4s) THEN
       #OrdenDato := 0;
       #Data_Addr := 43060;
   END_IF;
   IF (#Timer_LecturaMedidor.ET > t#4s) AND (#Timer_LecturaMedidor.ET < t#6s) THEN
       #OrdenDato := 1;
       #Data_Addr := 43068;
   END_IF;
END_REGION

REGION Network 3: Energias activa reactiva total
   RUNG wire#powerrail
      { S7_Templates := "SrcType := Time" } GT_Contact(in1 := #Timer_LecturaMedidor.ET, in2 := t#6s)
      { S7_Templates := "SrcType := Time" } LT_Contact(in1 := #Timer_LecturaMedidor.ET, in2 := t#8s)
      wire#w1
      Move(in := 2, out1 => #OrdenDato)
   END_RUNG
   RUNG wire#w1
      Move(in := 43059, out1 => #Data_Addr)
   END_RUNG
   RUNG wire#powerrail
      { S7_Templates := "SrcType := Time" } GT_Contact(in1 := #Timer_LecturaMedidor.ET, in2 := t#8s)
      { S7_Templates := "SrcType := Time" } LT_Contact(in1 := #Timer_LecturaMedidor.ET, in2 := t#10s)
      wire#w2
      Move(in := 3, out1 => #OrdenDato)
   END_RUNG
   RUNG wire#w2
      Move(in := 43067, out1 => #Data_Addr)
   END_RUNG
   // the same network as SCL:
   IF (#Timer_LecturaMedidor.ET > t#6s) AND (#Timer_LecturaMedidor.ET < t#8s) THEN
       #OrdenDato := 2;
       #Data_Addr := 43059;
   END_IF;
   IF (#Timer_LecturaMedidor.ET > t#8s) AND (#Timer_LecturaMedidor.ET < t#10s) THEN
       #OrdenDato := 3;
       #Data_Addr := 43067;
   END_IF;
END_REGION

REGION Network 4: Frecuencia y desbalance maximo de corriente
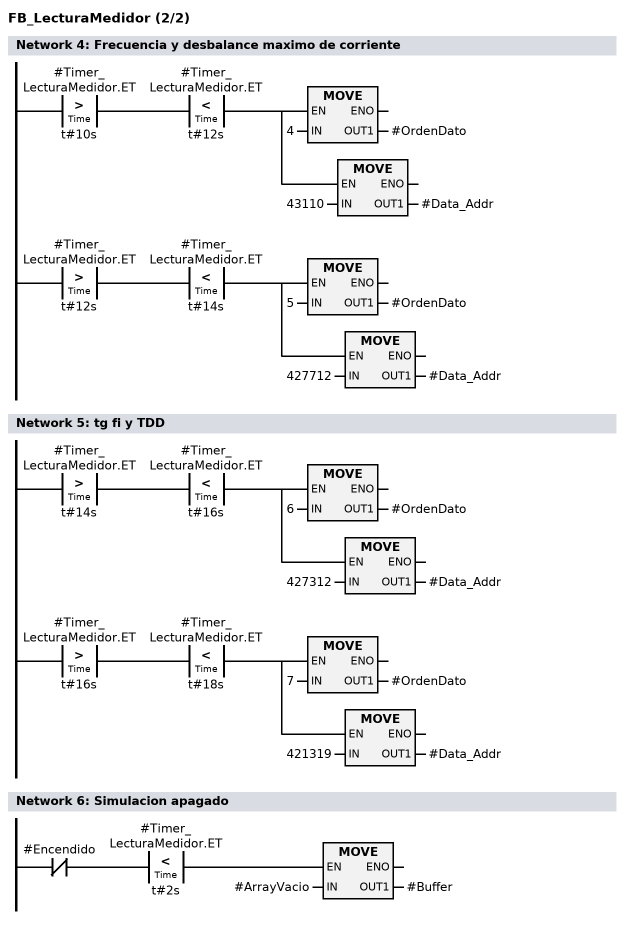
   RUNG wire#powerrail
      { S7_Templates := "SrcType := Time" } GT_Contact(in1 := #Timer_LecturaMedidor.ET, in2 := t#10s)
      { S7_Templates := "SrcType := Time" } LT_Contact(in1 := #Timer_LecturaMedidor.ET, in2 := t#12s)
      wire#w1
      Move(in := 4, out1 => #OrdenDato)
   END_RUNG
   RUNG wire#w1
      Move(in := 43110, out1 => #Data_Addr)
   END_RUNG
   RUNG wire#powerrail
      { S7_Templates := "SrcType := Time" } GT_Contact(in1 := #Timer_LecturaMedidor.ET, in2 := t#12s)
      { S7_Templates := "SrcType := Time" } LT_Contact(in1 := #Timer_LecturaMedidor.ET, in2 := t#14s)
      wire#w2
      Move(in := 5, out1 => #OrdenDato)
   END_RUNG
   RUNG wire#w2
      Move(in := 427712, out1 => #Data_Addr)
   END_RUNG
   // the same network as SCL:
   IF (#Timer_LecturaMedidor.ET > t#10s) AND (#Timer_LecturaMedidor.ET < t#12s) THEN
       #OrdenDato := 4;
       #Data_Addr := 43110;
   END_IF;
   IF (#Timer_LecturaMedidor.ET > t#12s) AND (#Timer_LecturaMedidor.ET < t#14s) THEN
       #OrdenDato := 5;
       #Data_Addr := 427712;
   END_IF;
END_REGION

REGION Network 5: tg fi y TDD
   RUNG wire#powerrail
      { S7_Templates := "SrcType := Time" } GT_Contact(in1 := #Timer_LecturaMedidor.ET, in2 := t#14s)
      { S7_Templates := "SrcType := Time" } LT_Contact(in1 := #Timer_LecturaMedidor.ET, in2 := t#16s)
      wire#w1
      Move(in := 6, out1 => #OrdenDato)
   END_RUNG
   RUNG wire#w1
      Move(in := 427312, out1 => #Data_Addr)
   END_RUNG
   RUNG wire#powerrail
      { S7_Templates := "SrcType := Time" } GT_Contact(in1 := #Timer_LecturaMedidor.ET, in2 := t#16s)
      { S7_Templates := "SrcType := Time" } LT_Contact(in1 := #Timer_LecturaMedidor.ET, in2 := t#18s)
      wire#w2
      Move(in := 7, out1 => #OrdenDato)
   END_RUNG
   RUNG wire#w2
      Move(in := 421319, out1 => #Data_Addr)
   END_RUNG
   // the same network as SCL:
   IF (#Timer_LecturaMedidor.ET > t#14s) AND (#Timer_LecturaMedidor.ET < t#16s) THEN
       #OrdenDato := 6;
       #Data_Addr := 427312;
   END_IF;
   IF (#Timer_LecturaMedidor.ET > t#16s) AND (#Timer_LecturaMedidor.ET < t#18s) THEN
       #OrdenDato := 7;
       #Data_Addr := 421319;
   END_IF;
END_REGION

REGION Network 6: Simulacion apagado
   RUNG wire#powerrail
      I_Contact( #Encendido )
      { S7_Templates := "SrcType := Time" } LT_Contact(in1 := #Timer_LecturaMedidor.ET, in2 := t#2s)
      Move(in := #ArrayVacio, out1 => #Buffer)
   END_RUNG
   // the same network as SCL:
   IF NOT #Encendido AND (#Timer_LecturaMedidor.ET < t#2s) THEN #Buffer := #ArrayVacio; END_IF;
END_REGION
END_FUNCTION_BLOCK

FUNCTION_BLOCK "FB_SimEmpacado"   // FB6, LAD
{ S7_Optimized_Access := 'TRUE' }
VERSION : 0.1
   VAR_INPUT
      Comando : Bool;
   END_VAR
   VAR_OUTPUT
      Mov : Int;
      Activada : Bool;
      Sentido : Int;
   END_VAR
   VAR
      EstadoComando : Bool;
      EstadoEmpacadora : Int;
      Timer_Apagado_Empacadora : TON_TIME;
   END_VAR
   VAR RETAIN
      ResetEmpacadora : Bool;
   END_VAR
   VAR
      ResetContajePositivo : Bool;
      TON_ContajePositivo : TON_TIME;
      Cajas : Int;
      ResetContajeNegativo : Bool;
      TON_ContajeNegativo : TON_TIME;
      ResetCajas : Bool;
   END_VAR
   VAR_TEMP   // added for the SCL form of the ladder/FBD networks
      _w1 : Bool;
      _w2 : Bool;
   END_VAR
BEGIN

REGION Network 1
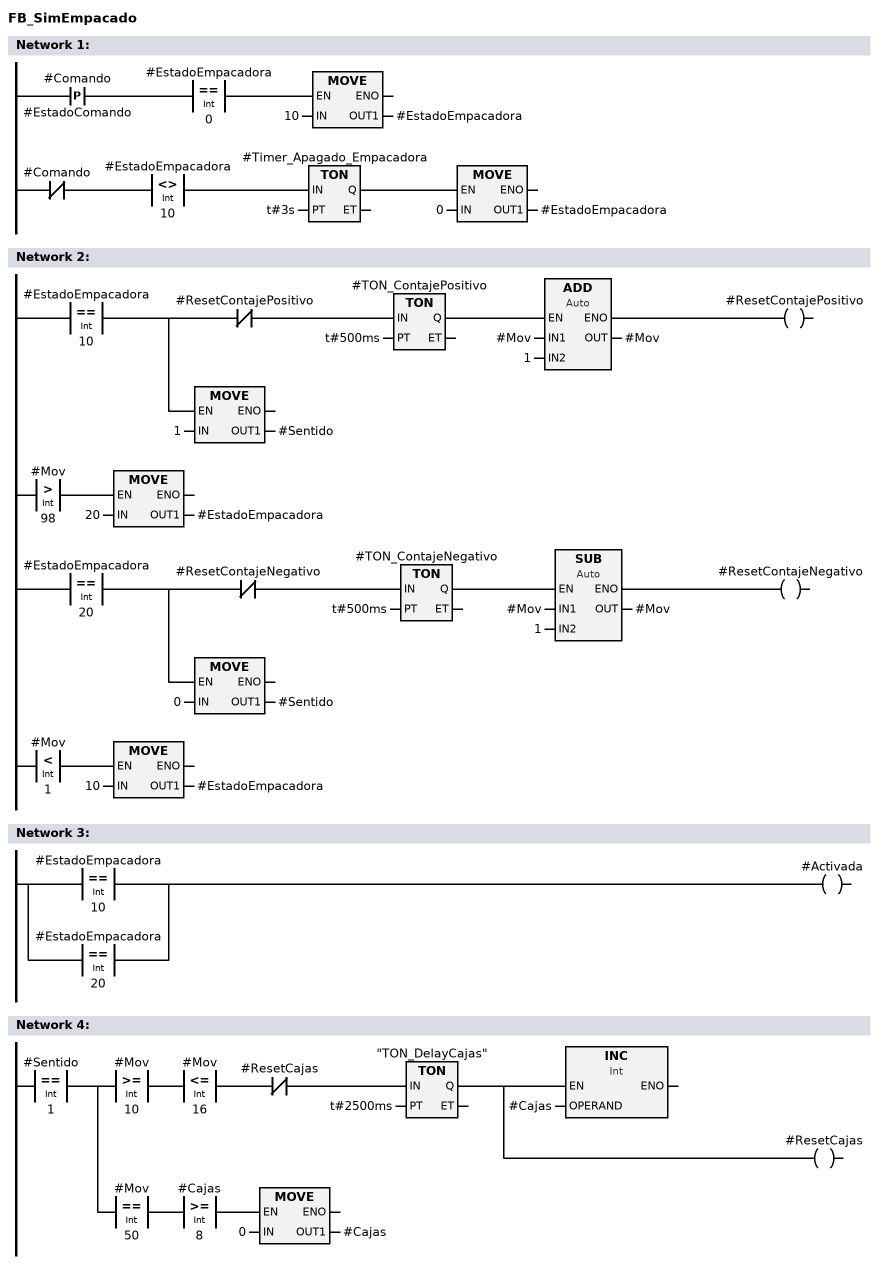
   #_w1 := #Comando AND NOT #EstadoComando;   // rising edge of #Comando
   #EstadoComando := #Comando;
   IF #_w1 AND (#EstadoEmpacadora = 0) THEN #EstadoEmpacadora := 10; END_IF;
   #Timer_Apagado_Empacadora(IN := NOT #Comando AND (#EstadoEmpacadora <> 10), PT := t#3s);   // TON
   IF #Timer_Apagado_Empacadora.Q THEN #EstadoEmpacadora := 0; END_IF;
END_REGION

REGION Network 2
   #_w1 := #EstadoEmpacadora = 10;
   #TON_ContajePositivo(IN := #_w1 AND NOT #ResetContajePositivo, PT := t#500ms);   // TON
   IF #TON_ContajePositivo.Q THEN #Mov := #Mov + 1; END_IF;
   #ResetContajePositivo := #TON_ContajePositivo.Q;
   IF #_w1 THEN #Sentido := 1; END_IF;
   IF #Mov > 98 THEN #EstadoEmpacadora := 20; END_IF;
   #_w2 := #EstadoEmpacadora = 20;
   #TON_ContajeNegativo(IN := #_w2 AND NOT #ResetContajeNegativo, PT := t#500ms);   // TON
   IF #TON_ContajeNegativo.Q THEN #Mov := #Mov - 1; END_IF;
   #ResetContajeNegativo := #TON_ContajeNegativo.Q;
   IF #_w2 THEN #Sentido := 0; END_IF;
   IF #Mov < 1 THEN #EstadoEmpacadora := 10; END_IF;
END_REGION

REGION Network 3
   RUNG wire#powerrail
      { S7_Templates := "SrcType := Int" } EQ_Contact(in1 := #EstadoEmpacadora, in2 := 10)
      wire#w1
      Coil( #Activada )
   END_RUNG
   RUNG wire#powerrail
      { S7_Templates := "SrcType := Int" } EQ_Contact(in1 := #EstadoEmpacadora, in2 := 20)
   END_RUNG wire#w1
   // the same network as SCL:
   #Activada := (#EstadoEmpacadora = 10) OR (#EstadoEmpacadora = 20);
END_REGION

REGION Network 4
   #_w1 := #Sentido = 1;
   "TON_DelayCajas".TON(IN := #_w1 AND (#Mov >= 10) AND (#Mov <= 16) AND NOT #ResetCajas, PT := t#2500ms);
   IF "TON_DelayCajas".Q THEN #Cajas := #Cajas + 1; END_IF;
   #ResetCajas := "TON_DelayCajas".Q;
   IF #_w1 AND (#Mov = 50) AND (#Cajas >= 8) THEN #Cajas := 0; END_IF;
END_REGION
END_FUNCTION_BLOCK

FUNCTION "FC_SimTensionPlanta" : Void   // FC1, LAD
{ S7_Optimized_Access := 'TRUE' }
VERSION : 0.1
   VAR_INPUT
      TensionL1 : Real;
      TensionL2 : Real;
      TensionL3 : Real;
   END_VAR
   VAR_OUTPUT
      TensionR1 : Real;
      TensionR2 : Real;
      TensionR3 : Real;
      TensionL1Escalada : Real;
      TensionL2Escalada : Real;
      TensionL3Escalada : Real;
      TensionR1Escalada : Real;
      TensionR2Escalada : Real;
      TensionR3Escalada : Real;
   END_VAR
   VAR_TEMP
      TensionAEscalarL1 : Real;
      TensionAEscalarL2 : Real;
      TensionAEscalarL3 : Real;
      TensionAEscalarR1 : Real;
      TensionAEscalarR2 : Real;
      TensionAEscalarR3 : Real;
   END_VAR
BEGIN

REGION Network 1
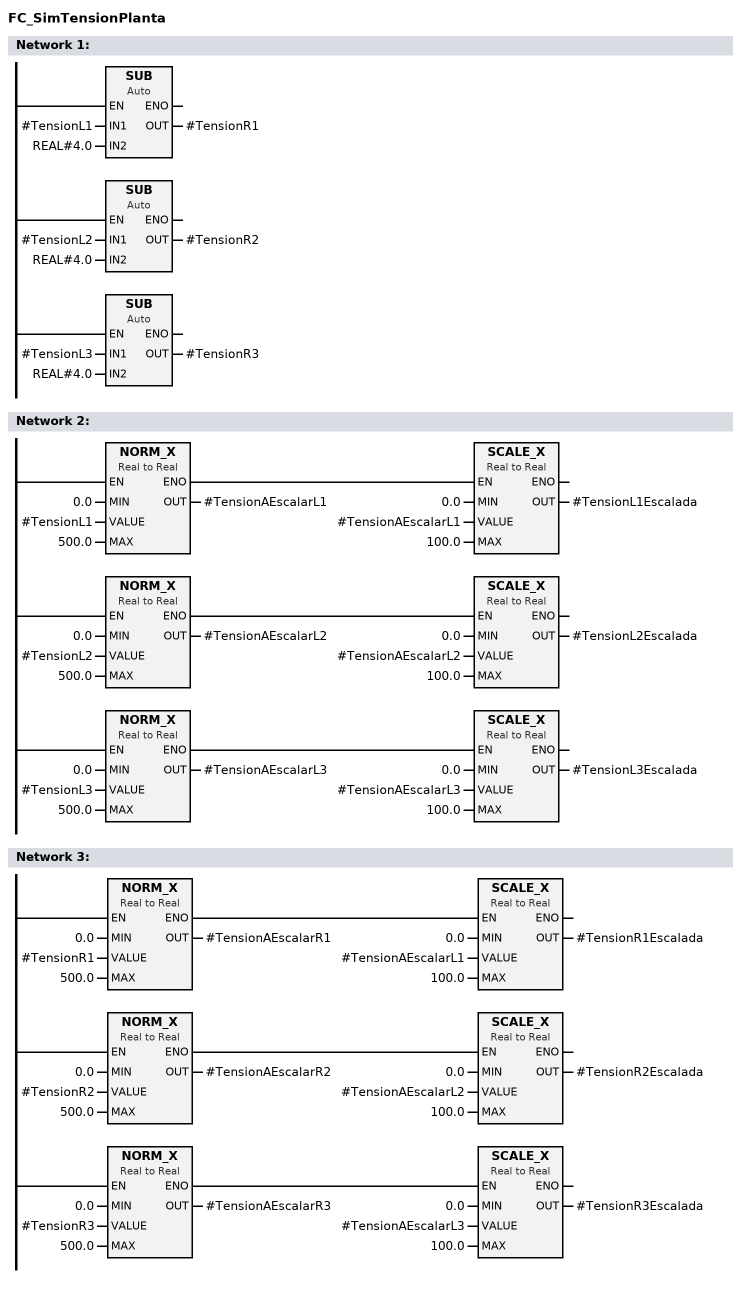
   RUNG wire#powerrail
      Sub(in1 := #TensionL1, in2 := REAL#4.0, out => #TensionR1)
   END_RUNG
   RUNG wire#powerrail
      Sub(in1 := #TensionL2, in2 := REAL#4.0, out => #TensionR2)
   END_RUNG
   RUNG wire#powerrail
      Sub(in1 := #TensionL3, in2 := REAL#4.0, out => #TensionR3)
   END_RUNG
   // the same network as SCL:
   #TensionR1 := #TensionL1 - REAL#4.0;
   #TensionR2 := #TensionL2 - REAL#4.0;
   #TensionR3 := #TensionL3 - REAL#4.0;
END_REGION

REGION Network 2
   RUNG wire#powerrail
      { S7_Templates := "[SrcType := Real, DestType := Real]" } Normalize(min := 0.0, value := #TensionL1, max := 500.0, out => #TensionAEscalarL1)
      { S7_Templates := "[SrcType := Real, DestType := Real]" } Scale(min := 0.0, value := #TensionAEscalarL1, max := 100.0, out => #TensionL1Escalada)
   END_RUNG
   RUNG wire#powerrail
      { S7_Templates := "[SrcType := Real, DestType := Real]" } Normalize(min := 0.0, value := #TensionL2, max := 500.0, out => #TensionAEscalarL2)
      { S7_Templates := "[SrcType := Real, DestType := Real]" } Scale(min := 0.0, value := #TensionAEscalarL2, max := 100.0, out => #TensionL2Escalada)
   END_RUNG
   RUNG wire#powerrail
      { S7_Templates := "[SrcType := Real, DestType := Real]" } Normalize(min := 0.0, value := #TensionL3, max := 500.0, out => #TensionAEscalarL3)
      { S7_Templates := "[SrcType := Real, DestType := Real]" } Scale(min := 0.0, value := #TensionAEscalarL3, max := 100.0, out => #TensionL3Escalada)
   END_RUNG
   // the same network as SCL:
   #TensionAEscalarL1 := NORM_X(MIN := 0.0, VALUE := #TensionL1, MAX := 500.0);
   #TensionL1Escalada := SCALE_X(MIN := 0.0, VALUE := #TensionAEscalarL1, MAX := 100.0);
   #TensionAEscalarL2 := NORM_X(MIN := 0.0, VALUE := #TensionL2, MAX := 500.0);
   #TensionL2Escalada := SCALE_X(MIN := 0.0, VALUE := #TensionAEscalarL2, MAX := 100.0);
   #TensionAEscalarL3 := NORM_X(MIN := 0.0, VALUE := #TensionL3, MAX := 500.0);
   #TensionL3Escalada := SCALE_X(MIN := 0.0, VALUE := #TensionAEscalarL3, MAX := 100.0);
END_REGION

REGION Network 3
   RUNG wire#powerrail
      { S7_Templates := "[SrcType := Real, DestType := Real]" } Normalize(min := 0.0, value := #TensionR1, max := 500.0, out => #TensionAEscalarR1)
      { S7_Templates := "[SrcType := Real, DestType := Real]" } Scale(min := 0.0, value := #TensionAEscalarL1, max := 100.0, out => #TensionR1Escalada)
   END_RUNG
   RUNG wire#powerrail
      { S7_Templates := "[SrcType := Real, DestType := Real]" } Normalize(min := 0.0, value := #TensionR2, max := 500.0, out => #TensionAEscalarR2)
      { S7_Templates := "[SrcType := Real, DestType := Real]" } Scale(min := 0.0, value := #TensionAEscalarL2, max := 100.0, out => #TensionR2Escalada)
   END_RUNG
   RUNG wire#powerrail
      { S7_Templates := "[SrcType := Real, DestType := Real]" } Normalize(min := 0.0, value := #TensionR3, max := 500.0, out => #TensionAEscalarR3)
      { S7_Templates := "[SrcType := Real, DestType := Real]" } Scale(min := 0.0, value := #TensionAEscalarL3, max := 100.0, out => #TensionR3Escalada)
   END_RUNG
   // the same network as SCL:
   #TensionAEscalarR1 := NORM_X(MIN := 0.0, VALUE := #TensionR1, MAX := 500.0);
   #TensionR1Escalada := SCALE_X(MIN := 0.0, VALUE := #TensionAEscalarL1, MAX := 100.0);
   #TensionAEscalarR2 := NORM_X(MIN := 0.0, VALUE := #TensionR2, MAX := 500.0);
   #TensionR2Escalada := SCALE_X(MIN := 0.0, VALUE := #TensionAEscalarL2, MAX := 100.0);
   #TensionAEscalarR3 := NORM_X(MIN := 0.0, VALUE := #TensionR3, MAX := 500.0);
   #TensionR3Escalada := SCALE_X(MIN := 0.0, VALUE := #TensionAEscalarL3, MAX := 100.0);
END_REGION
END_FUNCTION

ORGANIZATION_BLOCK "Main"   // OB1, LAD, ProgramCycle
{ S7_Optimized_Access := 'TRUE' }
VERSION : 0.1
   VAR_INPUT
      Initial_Call : Bool;
      Remanence : Bool;
   END_VAR
   VAR_TEMP   // added for the SCL form of the ladder/FBD networks
      _w1 : Bool;
      _w2 : Bool;
   END_VAR
BEGIN

REGION Network 1
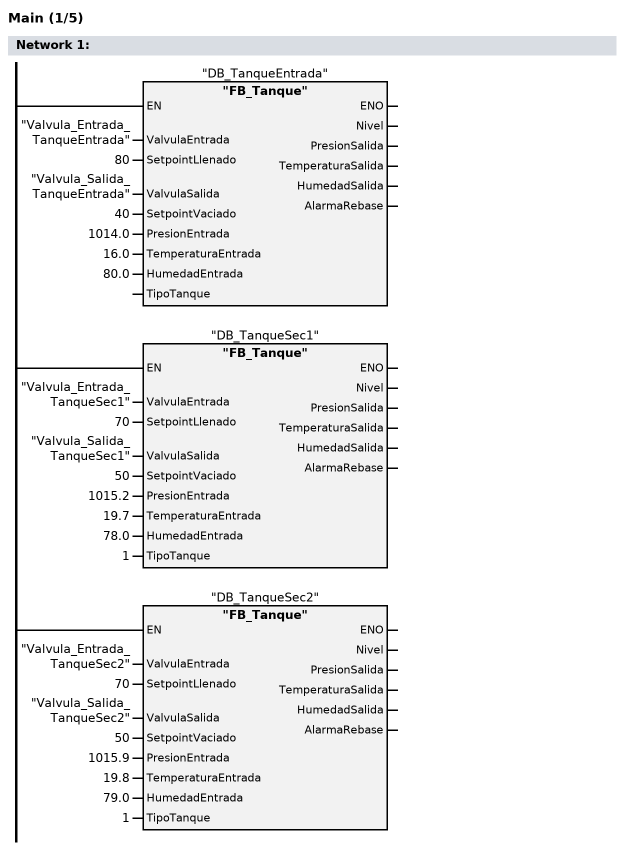
   RUNG wire#powerrail
      "DB_TanqueEntrada"(ValvulaEntrada := "Valvula_Entrada_TanqueEntrada", SetpointLlenado := 80, ValvulaSalida := "Valvula_Salida_TanqueEntrada", SetpointVaciado := 40, PresionEntrada := 1014.0, TemperaturaEntrada := 16.0, HumedadEntrada := 80.0, TipoTanque :=, Nivel =>, PresionSalida =>, TemperaturaSalida =>, HumedadSalida =>, AlarmaRebase =>)
   END_RUNG
   RUNG wire#powerrail
      "DB_TanqueSec1"(ValvulaEntrada := "Valvula_Entrada_TanqueSec1", SetpointLlenado := 70, ValvulaSalida := "Valvula_Salida_TanqueSec1", SetpointVaciado := 50, PresionEntrada := 1015.2, TemperaturaEntrada := 19.7, HumedadEntrada := 78.0, TipoTanque := 1, Nivel =>, PresionSalida =>, TemperaturaSalida =>, HumedadSalida =>, AlarmaRebase =>)
   END_RUNG
   RUNG wire#powerrail
      "DB_TanqueSec2"(ValvulaEntrada := "Valvula_Entrada_TanqueSec2", SetpointLlenado := 70, ValvulaSalida := "Valvula_Salida_TanqueSec2", SetpointVaciado := 50, PresionEntrada := 1015.9, TemperaturaEntrada := 19.8, HumedadEntrada := 79.0, TipoTanque := 1, Nivel =>, PresionSalida =>, TemperaturaSalida =>, HumedadSalida =>, AlarmaRebase =>)
   END_RUNG
   // the same network as SCL:
   "DB_TanqueEntrada"(ValvulaEntrada := "Valvula_Entrada_TanqueEntrada",   // "FB_Tanque"
                      SetpointLlenado := 80,
                      ValvulaSalida := "Valvula_Salida_TanqueEntrada",
                      SetpointVaciado := 40,
                      PresionEntrada := 1014.0,
                      TemperaturaEntrada := 16.0,
                      HumedadEntrada := 80.0);
   "DB_TanqueSec1"(ValvulaEntrada := "Valvula_Entrada_TanqueSec1",   // "FB_Tanque"
                   SetpointLlenado := 70,
                   ValvulaSalida := "Valvula_Salida_TanqueSec1",
                   SetpointVaciado := 50,
                   PresionEntrada := 1015.2,
                   TemperaturaEntrada := 19.7,
                   HumedadEntrada := 78.0,
                   TipoTanque := 1);
   "DB_TanqueSec2"(ValvulaEntrada := "Valvula_Entrada_TanqueSec2",   // "FB_Tanque"
                   SetpointLlenado := 70,
                   ValvulaSalida := "Valvula_Salida_TanqueSec2",
                   SetpointVaciado := 50,
                   PresionEntrada := 1015.9,
                   TemperaturaEntrada := 19.8,
                   HumedadEntrada := 79.0,
                   TipoTanque := 1);
END_REGION

REGION Network 2
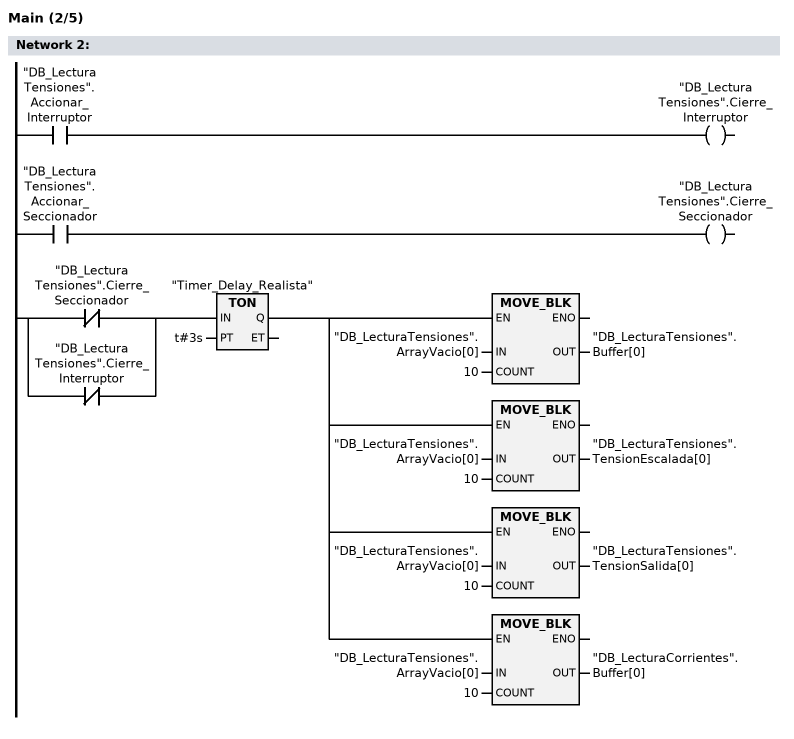
   "DB_LecturaTensiones".Cierre_Interruptor := "DB_LecturaTensiones".Accionar_Interruptor;
   "DB_LecturaTensiones".Cierre_Seccionador := "DB_LecturaTensiones".Accionar_Seccionador;
   "Timer_Delay_Realista".TON(IN := NOT "DB_LecturaTensiones".Cierre_Seccionador OR NOT "DB_LecturaTensiones".Cierre_Interruptor,
                           PT := t#3s);
   #_w1 := "Timer_Delay_Realista".Q;
   IF #_w1 THEN
       MOVE_BLK(IN := "DB_LecturaTensiones".ArrayVacio[0], COUNT := 10, OUT => "DB_LecturaTensiones".Buffer[0]);
       MOVE_BLK(IN := "DB_LecturaTensiones".ArrayVacio[0],
                COUNT := 10,
                OUT => "DB_LecturaTensiones".TensionEscalada[0]);
       MOVE_BLK(IN := "DB_LecturaTensiones".ArrayVacio[0],
                COUNT := 10,
                OUT => "DB_LecturaTensiones".TensionSalida[0]);
       MOVE_BLK(IN := "DB_LecturaTensiones".ArrayVacio[0], COUNT := 10, OUT => "DB_LecturaCorrientes".Buffer[0]);
   END_IF;
END_REGION

REGION Network 3
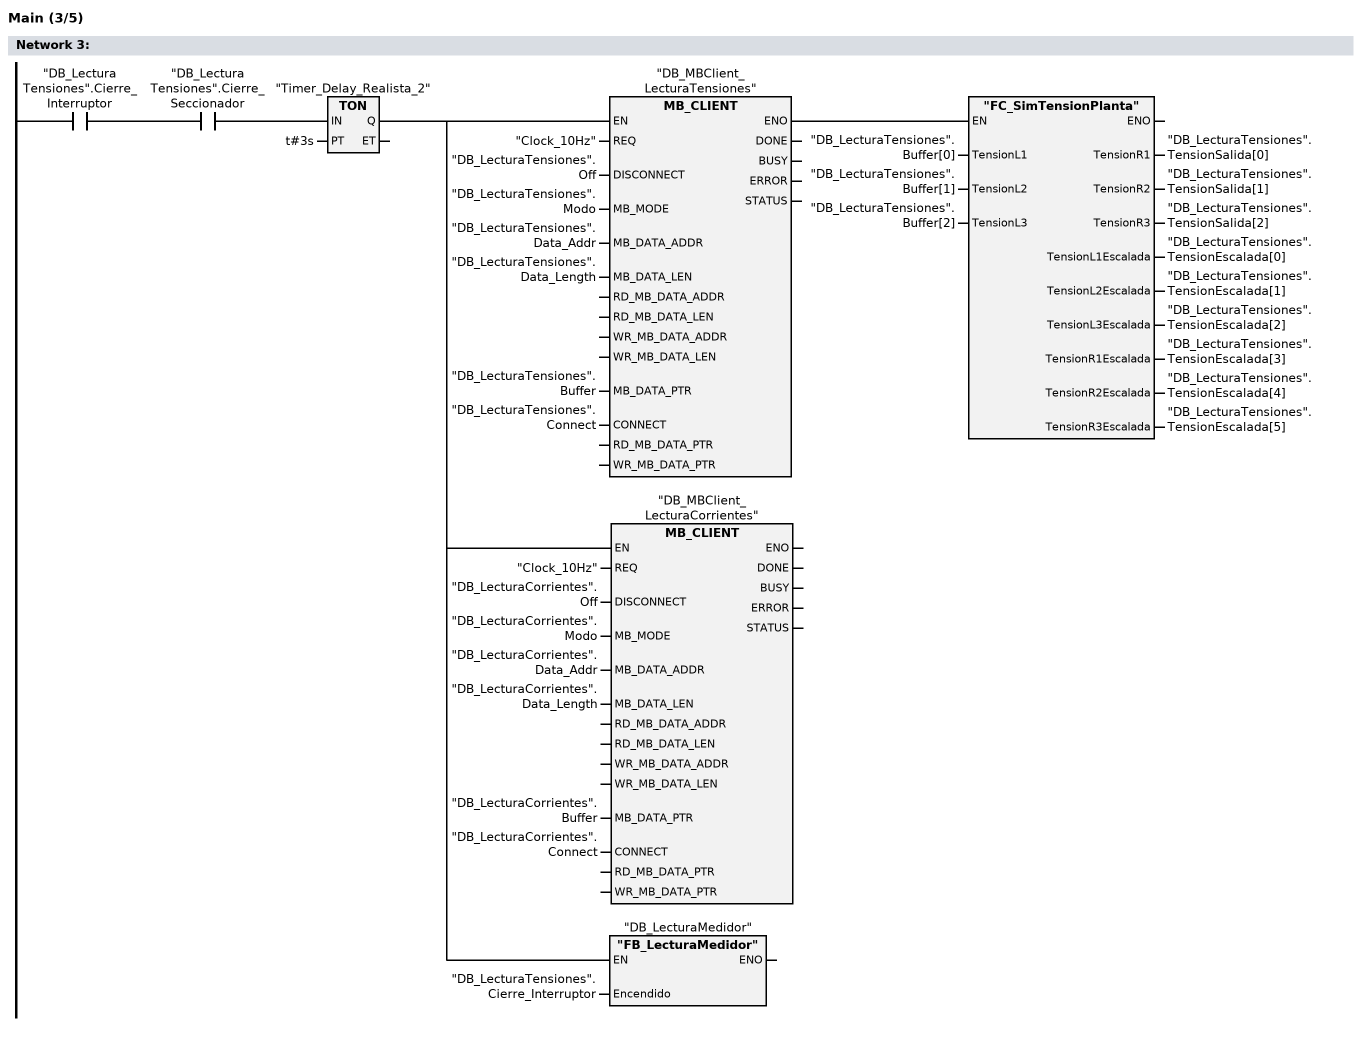
   // ENO of a box is taken as its EN; it also drops when the box reports an error
   "Timer_Delay_Realista_2".TON(IN := "DB_LecturaTensiones".Cierre_Interruptor AND "DB_LecturaTensiones".Cierre_Seccionador,
                           PT := t#3s);
   #_w1 := "Timer_Delay_Realista_2".Q;
   #_w2 := "Timer_Delay_Realista_2".Q;
   IF #_w2 THEN
       "DB_MBClient_LecturaTensiones"(REQ := "Clock_10Hz",   // MB_CLIENT
                               DISCONNECT := "DB_LecturaTensiones".Off,
                               MB_MODE := "DB_LecturaTensiones".Modo,
                               MB_DATA_ADDR := "DB_LecturaTensiones".Data_Addr,
                               MB_DATA_LEN := "DB_LecturaTensiones".Data_Length,
                               MB_DATA_PTR := "DB_LecturaTensiones".Buffer,
                               CONNECT := "DB_LecturaTensiones".Connect);
       "FC_SimTensionPlanta"(TensionL1 := "DB_LecturaTensiones".Buffer[0],
                             TensionL2 := "DB_LecturaTensiones".Buffer[1],
                             TensionL3 := "DB_LecturaTensiones".Buffer[2],
                             TensionR1 => "DB_LecturaTensiones".TensionSalida[0],
                             TensionR2 => "DB_LecturaTensiones".TensionSalida[1],
                             TensionR3 => "DB_LecturaTensiones".TensionSalida[2],
                             TensionL1Escalada => "DB_LecturaTensiones".TensionEscalada[0],
                             TensionL2Escalada => "DB_LecturaTensiones".TensionEscalada[1],
                             TensionL3Escalada => "DB_LecturaTensiones".TensionEscalada[2],
                             TensionR1Escalada => "DB_LecturaTensiones".TensionEscalada[3],
                             TensionR2Escalada => "DB_LecturaTensiones".TensionEscalada[4],
                             TensionR3Escalada => "DB_LecturaTensiones".TensionEscalada[5]);
   END_IF;
   IF #_w1 THEN
       "DB_MBClient_LecturaCorrientes"(REQ := "Clock_10Hz",   // MB_CLIENT
                               DISCONNECT := "DB_LecturaCorrientes".Off,
                               MB_MODE := "DB_LecturaCorrientes".Modo,
                               MB_DATA_ADDR := "DB_LecturaCorrientes".Data_Addr,
                               MB_DATA_LEN := "DB_LecturaCorrientes".Data_Length,
                               MB_DATA_PTR := "DB_LecturaCorrientes".Buffer,
                               CONNECT := "DB_LecturaCorrientes".Connect);
       "DB_LecturaMedidor"(Encendido := "DB_LecturaTensiones".Cierre_Interruptor);   // "FB_LecturaMedidor"
   END_IF;
END_REGION

REGION Network 4
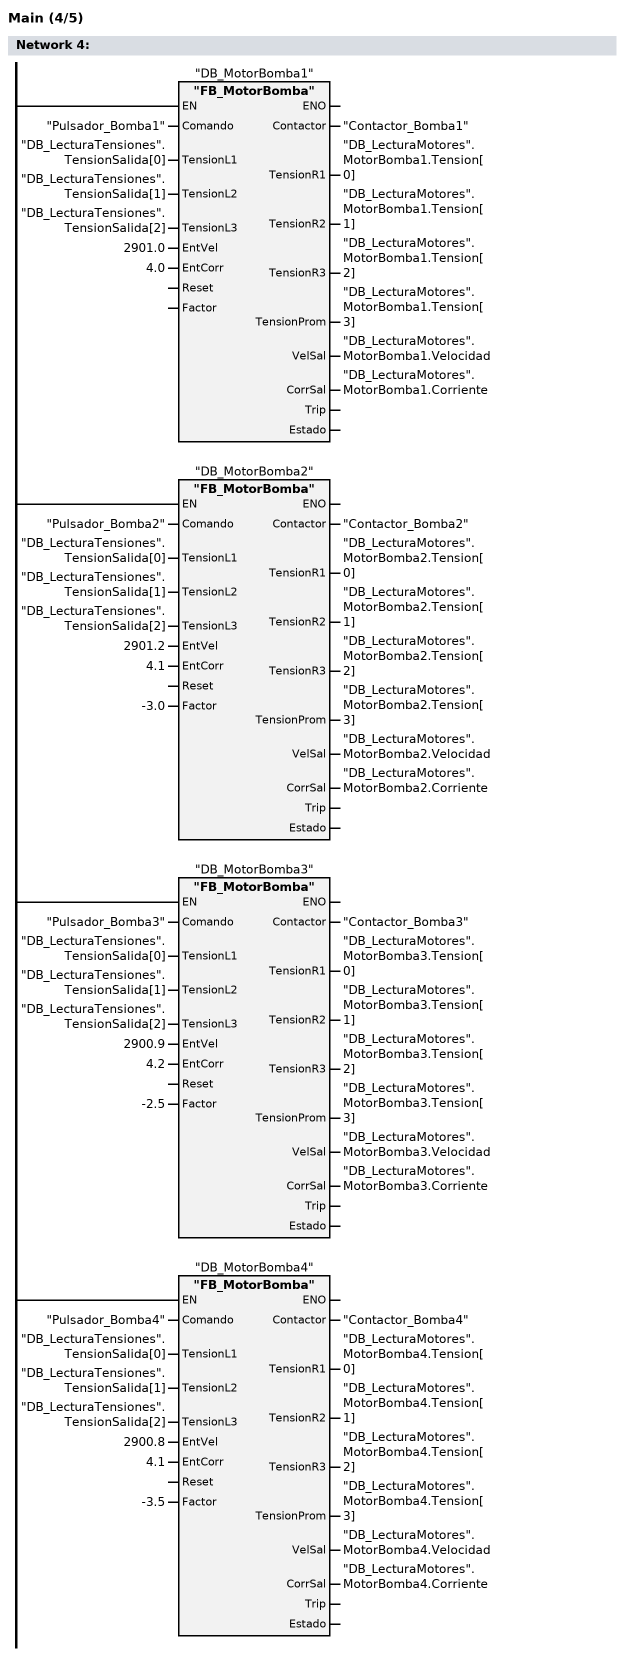
   RUNG wire#powerrail
      "DB_MotorBomba1"(Comando := "Pulsador_Bomba1", TensionL1 := "DB_LecturaTensiones".TensionSalida[0], TensionL2 := "DB_LecturaTensiones".TensionSalida[1], TensionL3 := "DB_LecturaTensiones".TensionSalida[2], EntVel := 2901.0, EntCorr := 4.0, Reset :=, Factor :=, Contactor => "Contactor_Bomba1", TensionR1 => "DB_LecturaMotores".MotorBomba1.Tension[0], TensionR2 => "DB_LecturaMotores".MotorBomba1.Tension[1], TensionR3 => "DB_LecturaMotores".MotorBomba1.Tension[2], TensionProm => "DB_LecturaMotores".MotorBomba1.Tension[3], VelSal => "DB_LecturaMotores".MotorBomba1.Velocidad, CorrSal => "DB_LecturaMotores".MotorBomba1.Corriente, Trip =>, Estado =>)
   END_RUNG
   RUNG wire#powerrail
      "DB_MotorBomba2"(Comando := "Pulsador_Bomba2", TensionL1 := "DB_LecturaTensiones".TensionSalida[0], TensionL2 := "DB_LecturaTensiones".TensionSalida[1], TensionL3 := "DB_LecturaTensiones".TensionSalida[2], EntVel := 2901.2, EntCorr := 4.1, Reset :=, Factor := -3.0, Contactor => "Contactor_Bomba2", TensionR1 => "DB_LecturaMotores".MotorBomba2.Tension[0], TensionR2 => "DB_LecturaMotores".MotorBomba2.Tension[1], TensionR3 => "DB_LecturaMotores".MotorBomba2.Tension[2], TensionProm => "DB_LecturaMotores".MotorBomba2.Tension[3], VelSal => "DB_LecturaMotores".MotorBomba2.Velocidad, CorrSal => "DB_LecturaMotores".MotorBomba2.Corriente, Trip =>, Estado =>)
   END_RUNG
   RUNG wire#powerrail
      "DB_MotorBomba3"(Comando := "Pulsador_Bomba3", TensionL1 := "DB_LecturaTensiones".TensionSalida[0], TensionL2 := "DB_LecturaTensiones".TensionSalida[1], TensionL3 := "DB_LecturaTensiones".TensionSalida[2], EntVel := 2900.9, EntCorr := 4.2, Reset :=, Factor := -2.5, Contactor => "Contactor_Bomba3", TensionR1 => "DB_LecturaMotores".MotorBomba3.Tension[0], TensionR2 => "DB_LecturaMotores".MotorBomba3.Tension[1], TensionR3 => "DB_LecturaMotores".MotorBomba3.Tension[2], TensionProm => "DB_LecturaMotores".MotorBomba3.Tension[3], VelSal => "DB_LecturaMotores".MotorBomba3.Velocidad, CorrSal => "DB_LecturaMotores".MotorBomba3.Corriente, Trip =>, Estado =>)
   END_RUNG
   RUNG wire#powerrail
      "DB_MotorBomba4"(Comando := "Pulsador_Bomba4", TensionL1 := "DB_LecturaTensiones".TensionSalida[0], TensionL2 := "DB_LecturaTensiones".TensionSalida[1], TensionL3 := "DB_LecturaTensiones".TensionSalida[2], EntVel := 2900.8, EntCorr := 4.1, Reset :=, Factor := -3.5, Contactor => "Contactor_Bomba4", TensionR1 => "DB_LecturaMotores".MotorBomba4.Tension[0], TensionR2 => "DB_LecturaMotores".MotorBomba4.Tension[1], TensionR3 => "DB_LecturaMotores".MotorBomba4.Tension[2], TensionProm => "DB_LecturaMotores".MotorBomba4.Tension[3], VelSal => "DB_LecturaMotores".MotorBomba4.Velocidad, CorrSal => "DB_LecturaMotores".MotorBomba4.Corriente, Trip =>, Estado =>)
   END_RUNG
   // the same network as SCL:
   "DB_MotorBomba1"(Comando := "Pulsador_Bomba1",   // "FB_MotorBomba"
                    TensionL1 := "DB_LecturaTensiones".TensionSalida[0],
                    TensionL2 := "DB_LecturaTensiones".TensionSalida[1],
                    TensionL3 := "DB_LecturaTensiones".TensionSalida[2],
                    EntVel := 2901.0,
                    EntCorr := 4.0,
                    Contactor => "Contactor_Bomba1",
                    TensionR1 => "DB_LecturaMotores".MotorBomba1.Tension[0],
                    TensionR2 => "DB_LecturaMotores".MotorBomba1.Tension[1],
                    TensionR3 => "DB_LecturaMotores".MotorBomba1.Tension[2],
                    TensionProm => "DB_LecturaMotores".MotorBomba1.Tension[3],
                    VelSal => "DB_LecturaMotores".MotorBomba1.Velocidad,
                    CorrSal => "DB_LecturaMotores".MotorBomba1.Corriente);
   "DB_MotorBomba2"(Comando := "Pulsador_Bomba2",   // "FB_MotorBomba"
                    TensionL1 := "DB_LecturaTensiones".TensionSalida[0],
                    TensionL2 := "DB_LecturaTensiones".TensionSalida[1],
                    TensionL3 := "DB_LecturaTensiones".TensionSalida[2],
                    EntVel := 2901.2,
                    EntCorr := 4.1,
                    Factor := -3.0,
                    Contactor => "Contactor_Bomba2",
                    TensionR1 => "DB_LecturaMotores".MotorBomba2.Tension[0],
                    TensionR2 => "DB_LecturaMotores".MotorBomba2.Tension[1],
                    TensionR3 => "DB_LecturaMotores".MotorBomba2.Tension[2],
                    TensionProm => "DB_LecturaMotores".MotorBomba2.Tension[3],
                    VelSal => "DB_LecturaMotores".MotorBomba2.Velocidad,
                    CorrSal => "DB_LecturaMotores".MotorBomba2.Corriente);
   "DB_MotorBomba3"(Comando := "Pulsador_Bomba3",   // "FB_MotorBomba"
                    TensionL1 := "DB_LecturaTensiones".TensionSalida[0],
                    TensionL2 := "DB_LecturaTensiones".TensionSalida[1],
                    TensionL3 := "DB_LecturaTensiones".TensionSalida[2],
                    EntVel := 2900.9,
                    EntCorr := 4.2,
                    Factor := -2.5,
                    Contactor => "Contactor_Bomba3",
                    TensionR1 => "DB_LecturaMotores".MotorBomba3.Tension[0],
                    TensionR2 => "DB_LecturaMotores".MotorBomba3.Tension[1],
                    TensionR3 => "DB_LecturaMotores".MotorBomba3.Tension[2],
                    TensionProm => "DB_LecturaMotores".MotorBomba3.Tension[3],
                    VelSal => "DB_LecturaMotores".MotorBomba3.Velocidad,
                    CorrSal => "DB_LecturaMotores".MotorBomba3.Corriente);
   "DB_MotorBomba4"(Comando := "Pulsador_Bomba4",   // "FB_MotorBomba"
                    TensionL1 := "DB_LecturaTensiones".TensionSalida[0],
                    TensionL2 := "DB_LecturaTensiones".TensionSalida[1],
                    TensionL3 := "DB_LecturaTensiones".TensionSalida[2],
                    EntVel := 2900.8,
                    EntCorr := 4.1,
                    Factor := -3.5,
                    Contactor => "Contactor_Bomba4",
                    TensionR1 => "DB_LecturaMotores".MotorBomba4.Tension[0],
                    TensionR2 => "DB_LecturaMotores".MotorBomba4.Tension[1],
                    TensionR3 => "DB_LecturaMotores".MotorBomba4.Tension[2],
                    TensionProm => "DB_LecturaMotores".MotorBomba4.Tension[3],
                    VelSal => "DB_LecturaMotores".MotorBomba4.Velocidad,
                    CorrSal => "DB_LecturaMotores".MotorBomba4.Corriente);
END_REGION

REGION Network 5
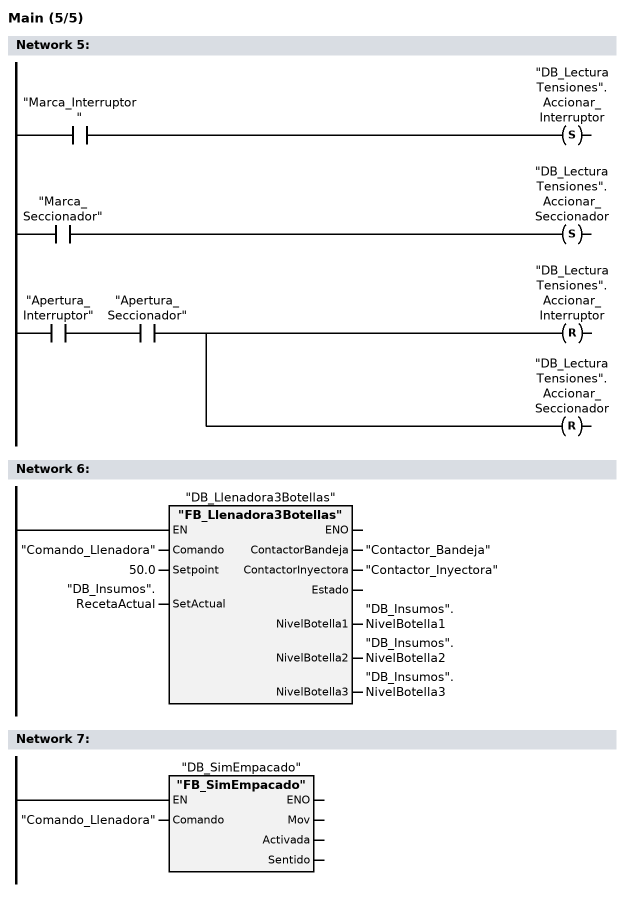
   RUNG wire#powerrail
      Contact( "Marca_Interruptor" )
      S_Coil( "DB_LecturaTensiones".Accionar_Interruptor )
   END_RUNG
   RUNG wire#powerrail
      Contact( "Marca_Seccionador" )
      S_Coil( "DB_LecturaTensiones".Accionar_Seccionador )
   END_RUNG
   RUNG wire#powerrail
      Contact( "Apertura_Interruptor" )
      Contact( "Apertura_Seccionador" )
      wire#w1
      R_Coil( "DB_LecturaTensiones".Accionar_Interruptor )
   END_RUNG
   RUNG wire#w1
      R_Coil( "DB_LecturaTensiones".Accionar_Seccionador )
   END_RUNG
   // the same network as SCL:
   IF "Marca_Interruptor" THEN "DB_LecturaTensiones".Accionar_Interruptor := TRUE; END_IF;
   IF "Marca_Seccionador" THEN "DB_LecturaTensiones".Accionar_Seccionador := TRUE; END_IF;
   IF "Apertura_Interruptor" AND "Apertura_Seccionador" THEN
       "DB_LecturaTensiones".Accionar_Interruptor := FALSE;
       "DB_LecturaTensiones".Accionar_Seccionador := FALSE;
   END_IF;
END_REGION

REGION Network 6
   RUNG wire#powerrail
      "DB_Llenadora3Botellas"(Comando := "Comando_Llenadora", Setpoint := 50.0, SetActual := "DB_Insumos".RecetaActual, ContactorBandeja => "Contactor_Bandeja", ContactorInyectora => "Contactor_Inyectora", Estado =>, NivelBotella1 => "DB_Insumos".NivelBotella1, NivelBotella2 => "DB_Insumos".NivelBotella2, NivelBotella3 => "DB_Insumos".NivelBotella3)
   END_RUNG
   // the same network as SCL:
   "DB_Llenadora3Botellas"(Comando := "Comando_Llenadora",   // "FB_Llenadora3Botellas"
                           Setpoint := 50.0,
                           SetActual := "DB_Insumos".RecetaActual,
                           ContactorBandeja => "Contactor_Bandeja",
                           ContactorInyectora => "Contactor_Inyectora",
                           NivelBotella1 => "DB_Insumos".NivelBotella1,
                           NivelBotella2 => "DB_Insumos".NivelBotella2,
                           NivelBotella3 => "DB_Insumos".NivelBotella3);
END_REGION

REGION Network 7
   RUNG wire#powerrail
      "DB_SimEmpacado"(Comando := "Comando_Llenadora", Mov =>, Activada =>, Sentido =>)
   END_RUNG
   // the same network as SCL:
   "DB_SimEmpacado"(Comando := "Comando_Llenadora");   // "FB_SimEmpacado"
END_REGION
END_ORGANIZATION_BLOCK